KUKA KRL program: MyProgram_150().src

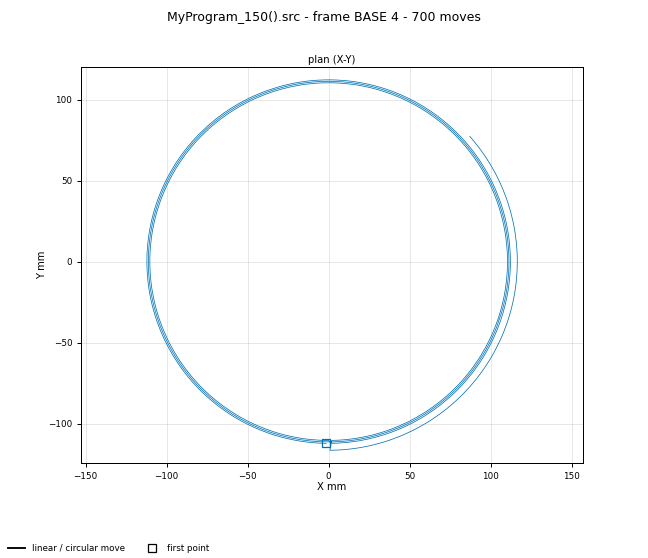
[picture p0: tool path of MyProgram_150().src in frame BASE 4, 700 of 700 moves have a stored position in this frame; points joined in program order, loops and branches not executed]
&ACCESS RVP
&REL 1
&PARAM TEMPLATE = C:\KRC\Roboter\Template\vorgabe
&PARAM EDITMASK = *
DEF MyProgram_150()
; ---- Setting reference (Base) ----
$BASE = BASE_DATA[4]

; --------------------------
; ---- Setting tool (TCP) ----
$TOOL = TOOL_DATA[3]
; --------------------------

$VEL.CP = VEL_APROX_PRINT
Startdeposition()
$VEL.CP = VEL_PRINT
LIN {X -1.5125,Y -112.2052,Z 117,A -94.956,B 24.9546,C -1.5569,E1 24.9968,E2 180.9074} C_DIS
LIN {X -5.7885,Y -112.0653,Z 117,A -97.1016,B 24.9546,C -1.5583,E1 24.9908,E2 183.05} C_DIS
LIN {X -9.0238,Y -111.8506,Z 117,A -99.1979,B 24.9556,C -1.5398,E1 24.9848,E2 185.1911} C_DIS
LIN {X -12.7167,Y -111.4916,Z 117,A -100.657,B 24.9545,C -1.5583,E1 24.9809,E2 186.6072} C_DIS
LIN {X -17.0349,Y -110.9135,Z 117,A -102.8531,B 24.9545,C -1.56,E1 24.9748,E2 188.801} C_DIS
LIN {X -20.6022,Y -110.3083,Z 117,A -104.7565,B 24.9545,C -1.5583,E1 24.9696,E2 190.7105} C_DIS
LIN {X -25.8364,Y -109.2008,Z 117,A -107.366,B 24.9541,C -1.5646,E1 24.9625,E2 193.3082} C_DIS
LIN {X -29.1128,Y -108.3718,Z 117,A -109.2021,B 24.9543,C -1.5611,E1 24.9575,E2 195.1553} C_DIS
LIN {X -32.9964,Y -107.2534,Z 117,A -111.2303,B 24.9542,C -1.564,E1 24.9521,E2 197.18} C_DIS
LIN {X -36.1753,Y -106.2236,Z 117,A -112.94,B 24.9541,C -1.5652,E1 24.9476,E2 198.89} C_DIS
LIN {X -41.7306,Y -104.1678,Z 117,A -116.2554,B 24.9546,C -1.5561,E1 24.9388,E2 202.2341} C_DIS
LIN {X -46.6403,Y -102.0638,Z 117,A -118.7805,B 24.954,C -1.5674,E1 24.9324,E2 204.7384} C_DIS
LIN {X -49.8054,Y -100.5555,Z 117,A -120.8158,B 24.9544,C -1.5596,E1 24.9273,E2 206.7975} C_DIS
LIN {X -53.3163,Y -98.739,Z 117,A -122.531,B 24.9535,C -1.5746,E1 24.9231,E2 208.4819} C_DIS
LIN {X -56.3522,Y -97.0395,Z 117,A -124.7681,B 24.9545,C -1.5584,E1 24.9176,E2 210.7639} C_DIS
LIN {X -59.4233,Y -95.1885,Z 117,A -125.8907,B 24.9526,C -1.5899,E1 24.9151,E2 211.8152} C_DIS
LIN {X -61.8008,Y -93.6624,Z 117,A -127.5917,B 24.9531,C -1.5817,E1 24.911,E2 213.5414} C_DIS
LIN {X -66.4782,Y -90.4029,Z 117,A -130.4958,B 24.9528,C -1.5868,E1 24.9044,E2 216.4431} C_DIS
LIN {X -69.3755,Y -88.1992,Z 117,A -132.4481,B 24.9528,C -1.5864,E1 24.9001,E2 218.4035} C_DIS
LIN {X -72.4947,Y -85.6542,Z 117,A -134.4851,B 24.9526,C -1.5911,E1 24.8957,E2 220.4373} C_DIS
LIN {X -75.0296,Y -83.4422,Z 117,A -136.1776,B 24.9523,C -1.5955,E1 24.8922,E2 222.126} C_DIS
LIN {X -79.2176,Y -79.4784,Z 117,A -139.0952,B 24.9519,C -1.6027,E1 24.8863,E2 225.0385} C_DIS
LIN {X -81.6863,Y -76.9372,Z 117,A -141.3411,B 24.9527,C -1.5894,E1 24.8819,E2 227.3258} C_DIS
LIN {X -84.0515,Y -74.349,Z 117,A -142.6578,B 24.9513,C -1.6121,E1 24.8796,E2 228.5943} C_DIS
LIN {X -86.8434,Y -71.0668,Z 117,A -145.025,B 24.9513,C -1.6107,E1 24.8753,E2 230.9758} C_DIS
LIN {X -89.0383,Y -68.2951,Z 117,A -146.8336,B 24.9511,C -1.6149,E1 24.8722,E2 232.7828} C_DIS
LIN {X -91.2603,Y -65.2959,Z 117,A -148.6799,B 24.9507,C -1.6221,E1 24.8692,E2 234.6212} C_DIS
LIN {X -93.1631,Y -62.5525,Z 117,A -150.6796,B 24.9511,C -1.6148,E1 24.866,E2 236.648} C_DIS
LIN {X -96.2181,Y -57.7447,Z 117,A -153.4338,B 24.9503,C -1.6285,E1 24.862,E2 239.3836} C_DIS
LIN {X -98.0482,Y -54.5762,Z 117,A -155.8431,B 24.9513,C -1.6126,E1 24.8586,E2 241.8434} C_DIS
LIN {X -100.1395,Y -50.6388,Z 117,A -157.3726,B 24.9491,C -1.648,E1 24.8568,E2 243.2969} C_DIS
LIN {X -101.3521,Y -48.166,Z 117,A -158.8369,B 24.9491,C -1.6497,E1 24.855,E2 244.7651} C_DIS
LIN {X -102.7604,Y -45.0816,Z 117,A -160.6671,B 24.9489,C -1.6508,E1 24.8529,E2 246.6026} C_DIS
LIN {X -104.005,Y -42.1305,Z 117,A -162.302,B 24.9486,C -1.6556,E1 24.8511,E2 248.2352} C_DIS
LIN {X -105.7444,Y -37.5537,Z 117,A -164.6186,B 24.9477,C -1.6701,E1 24.8489,E2 250.5302} C_DIS
LIN {X -106.8716,Y -34.2124,Z 117,A -166.8469,B 24.9484,C -1.659,E1 24.8469,E2 252.7979} C_DIS
LIN {X -108.0632,Y -30.2401,Z 117,A -168.866,B 24.9478,C -1.6692,E1 24.8453,E2 254.8042} C_DIS
LIN {X -108.9967,Y -26.6779,Z 117,A -170.6645,B 24.9472,C -1.6782,E1 24.8441,E2 256.5917} C_DIS
LIN {X -109.7546,Y -23.3715,Z 117,A -172.4769,B 24.9471,C -1.6805,E1 24.843,E2 258.4094} C_DIS
LIN {X -110.4905,Y -19.5938,Z 117,A -174.4741,B 24.9468,C -1.6855,E1 24.842,E2 260.4065} C_DIS
LIN {X -111.1169,Y -15.6532,Z 117,A -176.3681,B 24.946,C -1.6975,E1 24.8412,E2 262.2832} C_DIS
LIN {X -111.5012,Y -12.6345,Z 117,A -178.0918,B 24.9461,C -1.6959,E1 24.8407,E2 264.021} C_DIS
LIN {X -111.8621,Y -8.8796,Z 117,A -179.9252,B 24.9455,C -1.7057,E1 24.8402,E2 265.8421} C_DIS
LIN {X -112.1042,Y -4.9643,Z 117,A 178.0019,B 24.9452,C -1.7094,E1 24.8399,E2 267.9185} C_DIS
LIN {X -112.2093,Y -1.0958,Z 117,A 176.0457,B 24.9448,C -1.7166,E1 24.8398,E2 269.8693} C_DIS
LIN {X -112.1374,Y 4.1928,Z 117,A 173.4446,B 24.944,C -1.7292,E1 24.8399,E2 272.4561} C_DIS
LIN {X -112.0034,Y 6.9038,Z 117,A 171.8392,B 24.9442,C -1.7252,E1 24.8402,E2 274.0806} C_DIS
LIN {X -111.7118,Y 10.6091,Z 117,A 169.9421,B 24.9438,C -1.7315,E1 24.8406,E2 275.9742} C_DIS
LIN {X -111.2466,Y 14.7055,Z 117,A 167.8342,B 24.9434,C -1.7382,E1 24.8414,E2 278.0787} C_DIS
LIN {X -110.6476,Y 18.6849,Z 117,A 165.8922,B 24.9427,C -1.7492,E1 24.8422,E2 280.0061} C_DIS
LIN {X -109.9711,Y 22.3248,Z 117,A 163.9291,B 24.9424,C -1.7525,E1 24.8432,E2 281.9729} C_DIS
LIN {X -109.2275,Y 25.721,Z 117,A 162.069,B 24.9423,C -1.7549,E1 24.8444,E2 283.8381} C_DIS
LIN {X -108.2907,Y 29.4132,Z 117,A 160.2595,B 24.9415,C -1.7663,E1 24.8457,E2 285.6309} C_DIS
LIN {X -107.357,Y 32.662,Z 117,A 158.2689,B 24.9418,C -1.7616,E1 24.8473,E2 287.6443} C_DIS
LIN {X -106.3302,Y 35.8592,Z 117,A 156.7529,B 24.941,C -1.7747,E1 24.8486,E2 289.1378} C_DIS
LIN {X -105.2682,Y 38.8689,Z 117,A 155.1631,B 24.9405,C -1.7813,E1 24.8501,E2 290.7209} C_DIS
LIN {X -104.0689,Y 41.9735,Z 117,A 153.3117,B 24.9405,C -1.7807,E1 24.852,E2 292.584} C_DIS
LIN {X -102.6445,Y 45.3475,Z 117,A 150.7978,B 24.9418,C -1.7617,E1 24.8549,E2 295.1569} C_DIS
LIN {X -100.6823,Y 49.5496,Z 117,A 149.0628,B 24.9397,C -1.7931,E1 24.8569,E2 296.8266} C_DIS
LIN {X -98.9283,Y 52.9675,Z 117,A 147.0344,B 24.9395,C -1.7963,E1 24.8595,E2 298.8581} C_DIS
LIN {X -97.1624,Y 56.1383,Z 117,A 145.3017,B 24.9388,C -1.8064,E1 24.8619,E2 300.5758} C_DIS
LIN {X -95.2496,Y 59.3256,Z 117,A 143.0052,B 24.9395,C -1.7965,E1 24.8653,E2 302.9078} C_DIS
LIN {X -93.486,Y 62.0683,Z 117,A 141.5329,B 24.9387,C -1.8086,E1 24.8675,E2 304.3585} C_DIS
LIN {X -91.6074,Y 64.8095,Z 117,A 139.9194,B 24.9382,C -1.8165,E1 24.8701,E2 305.9611} C_DIS
LIN {X -89.6293,Y 67.5174,Z 117,A 137.734,B 24.9391,C -1.8029,E1 24.8739,E2 308.1894} C_DIS
LIN {X -87.2066,Y 70.6186,Z 117,A 136.2751,B 24.9373,C -1.8295,E1 24.8763,E2 309.5917} C_DIS
LIN {X -83.2861,Y 75.204,Z 117,A 133.3752,B 24.9362,C -1.8445,E1 24.8816,E2 312.469} C_DIS
LIN {X -80.5138,Y 78.1644,Z 117,A 130.8616,B 24.9371,C -1.8324,E1 24.8865,E2 315.0226} C_DIS
LIN {X -74.6442,Y 83.7873,Z 117,A 126.8667,B 24.936,C -1.8483,E1 24.8945,E2 318.9959} C_DIS
LIN {X -70.5545,Y 87.2586,Z 117,A 124.4485,B 24.9347,C -1.867,E1 24.8996,E2 321.3788} C_DIS
LIN {X -67.8838,Y 89.354,Z 117,A 122.5036,B 24.935,C -1.8623,E1 24.904,E2 323.342} C_DIS
LIN {X -64.7113,Y 91.6774,Z 117,A 119.9198,B 24.9363,C -1.8438,E1 24.9099,E2 325.9789} C_DIS
LIN {X -61.7752,Y 93.6793,Z 117,A 118.5231,B 24.9349,C -1.8638,E1 24.9131,E2 327.3326} C_DIS
LIN {X -58.5579,Y 95.7239,Z 117,A 116.5933,B 24.9346,C -1.8681,E1 24.9176,E2 329.2582} C_DIS
LIN {X -55.8629,Y 97.3207,Z 117,A 115.0159,B 24.9343,C -1.8719,E1 24.9214,E2 330.8313} C_DIS
LIN {X -52.9912,Y 98.9154,Z 117,A 112.7947,B 24.9356,C -1.8532,E1 24.927,E2 333.1033} C_DIS
LIN {X -49.5821,Y 100.6662,Z 117,A 111.2451,B 24.9343,C -1.8725,E1 24.9308,E2 334.611} C_DIS
LIN {X -45.8433,Y 102.4229,Z 117,A 108.3059,B 24.9363,C -1.8428,E1 24.9385,E2 337.628} C_DIS
LIN {X -40.6091,Y 104.6092,Z 117,A 106.523,B 24.933,C -1.8912,E1 24.9428,E2 339.2998} C_DIS
LIN {X -38.2643,Y 105.4887,Z 117,A 105.0656,B 24.9333,C -1.8857,E1 24.9467,E2 340.7734} C_DIS
LIN {X -30.9788,Y 107.8539,Z 117,A 101.3274,B 24.9325,C -1.8972,E1 24.9566,E2 344.4908} C_DIS
LIN {X -28.4362,Y 108.5525,Z 117,A 99.6995,B 24.9332,C -1.8871,E1 24.961,E2 346.1451} C_DIS
LIN {X -25.1714,Y 109.3544,Z 117,A 97.9354,B 24.9332,C -1.8868,E1 24.9658,E2 347.9122} C_DIS
LIN {X -21.2376,Y 110.186,Z 117,A 96.0146,B 24.9328,C -1.8939,E1 24.971,E2 349.8184} C_DIS
LIN {X -18.1728,Y 110.7332,Z 117,A 94.4475,B 24.9326,C -1.896,E1 24.9753,E2 351.382} C_DIS
LIN {X -13.9046,Y 111.3504,Z 117,A 92.3061,B 24.9323,C -1.8999,E1 24.9812,E2 353.516} C_DIS
LIN {X -9.8507,Y 111.7818,Z 117,A 90.2123,B 24.9323,C -1.9005,E1 24.9871,E2 355.6095} C_DIS
LIN {X -7.0871,Y 111.991,Z 117,A 88.5994,B 24.9328,C -1.8929,E1 24.9916,E2 357.241} C_DIS
LIN {X -2.0943,Y 112.1945,Z 117,A 85.7771,B 24.9336,C -1.8825,E1 24.9996,E2 360.0883} C_DIS
LIN {X 1.2742,Y 112.2083,Z 117,A 84.6091,B 24.9319,C -1.9057,E1 25.0027,E2 361.2014} C_DIS
LIN {X 4.8323,Y 112.1099,Z 117,A 82.6215,B 24.9324,C -1.8988,E1 25.0083,E2 363.2049} C_DIS
LIN {X 9.5577,Y 111.8079,Z 117,A 80.214,B 24.9324,C -1.8991,E1 25.015,E2 365.6106} C_DIS
LIN {X 13.3506,Y 111.4174,Z 117,A 78.1427,B 24.9328,C -1.8936,E1 25.0207,E2 367.6934} C_DIS
LIN {X 17.2419,Y 110.8815,Z 117,A 76.2936,B 24.9324,C -1.8996,E1 25.0258,E2 369.5266} C_DIS
LIN {X 20.1907,Y 110.3831,Z 117,A 74.6472,B 24.9328,C -1.894,E1 25.0304,E2 371.1845} C_DIS
LIN {X 24.2884,Y 109.5546,Z 117,A 72.4808,B 24.9329,C -1.8916,E1 25.0363,E2 373.3538} C_DIS
LIN {X 28.0609,Y 108.6489,Z 117,A 70.6583,B 24.9325,C -1.8972,E1 25.0412,E2 375.1604} C_DIS
LIN {X 31.3668,Y 107.7425,Z 117,A 68.7397,B 24.9331,C -1.8888,E1 25.0464,E2 377.0957} C_DIS
LIN {X 35.0187,Y 106.6111,Z 117,A 66.4582,B 24.9342,C -1.8733,E1 25.0525,E2 379.4097} C_DIS
LIN {X 38.3665,Y 105.4514,Z 117,A 65.4478,B 24.9319,C -1.9057,E1 25.055,E2 380.3413} C_DIS
LIN {X 41.2551,Y 104.3554,Z 117,A 63.4643,B 24.9333,C -1.8867,E1 25.0603,E2 382.3654} C_DIS
LIN {X 44.747,Y 102.9063,Z 117,A 61.6337,B 24.9331,C -1.8889,E1 25.0649,E2 384.1865} C_DIS
LIN {X 49.1094,Y 100.8988,Z 117,A 59.3592,B 24.9328,C -1.8936,E1 25.0707,E2 386.4441} C_DIS
LIN {X 52.9738,Y 98.9248,Z 117,A 55.9431,B 24.9366,C -1.8391,E1 25.0794,E2 389.9793} C_DIS
LIN {X 58.1394,Y 95.9782,Z 117,A 54.0163,B 24.9336,C -1.8823,E1 25.0838,E2 391.798} C_DIS
LIN {X 62.8187,Y 92.9828,Z 117,A 51.1015,B 24.9341,C -1.8744,E1 25.0906,E2 394.7221} C_DIS
LIN {X 65.5667,Y 91.0671,Z 117,A 49.3016,B 24.9346,C -1.8675,E1 25.0947,E2 396.532} C_DIS
LIN {X 68.3874,Y 88.9672,Z 117,A 47.564,B 24.9346,C -1.8668,E1 25.0986,E2 398.2649} C_DIS
LIN {X 71.2508,Y 86.693,Z 117,A 45.6537,B 24.9351,C -1.8614,E1 25.1027,E2 400.1809} C_DIS
LIN {X 74.0379,Y 84.3236,Z 117,A 42.9238,B 24.9379,C -1.8201,E1 25.1087,E2 402.9974} C_DIS
LIN {X 78.3419,Y 80.3427,Z 117,A 40.982,B 24.9352,C -1.8598,E1 25.1124,E2 404.8375} C_DIS
LIN {X 82.243,Y 76.3446,Z 117,A 38.1481,B 24.9355,C -1.8543,E1 25.1179,E2 407.6722} C_DIS
LIN {X 84.3331,Y 74.0269,Z 117,A 36.4291,B 24.9362,C -1.8451,E1 25.1211,E2 409.4052} C_DIS
LIN {X 86.6293,Y 71.3275,Z 117,A 34.2171,B 24.9377,C -1.823,E1 25.1251,E2 411.6592} C_DIS
LIN {X 88.8607,Y 68.5257,Z 117,A 32.8714,B 24.9365,C -1.8399,E1 25.1273,E2 412.9585} C_DIS
LIN {X 91.0579,Y 65.5797,Z 117,A 30.8711,B 24.9372,C -1.8297,E1 25.1306,E2 414.9733} C_DIS
LIN {X 93.2181,Y 62.4712,Z 117,A 28.7974,B 24.938,C -1.8185,E1 25.1339,E2 417.0633} C_DIS
LIN {X 95.3528,Y 59.1603,Z 117,A 26.9952,B 24.9377,C -1.8225,E1 25.1366,E2 418.847} C_DIS
LIN {X 97.6683,Y 55.2565,Z 117,A 24.8595,B 24.9377,C -1.8243,E1 25.1396,E2 420.9673} C_DIS
LIN {X 99.1265,Y 52.5931,Z 117,A 23.2054,B 24.9382,C -1.8154,E1 25.1418,E2 422.6338} C_DIS
LIN {X 100.6594,Y 49.5957,Z 117,A 21.0654,B 24.9398,C -1.7917,E1 25.1445,E2 424.8181} C_DIS
LIN {X 102.2017,Y 46.3343,Z 117,A 19.95,B 24.938,C -1.8191,E1 25.1457,E2 425.8631} C_DIS
LIN {X 103.3763,Y 43.65,Z 117,A 18.0055,B 24.9396,C -1.7945,E1 25.1479,E2 427.8548} C_DIS
LIN {X 105.4616,Y 38.3386,Z 117,A 15.2835,B 24.9396,C -1.7945,E1 25.1506,E2 430.5617} C_DIS
LIN {X 106.7401,Y 34.6199,Z 117,A 13.2706,B 24.9401,C -1.7882,E1 25.1524,E2 432.578} C_DIS
LIN {X 107.7174,Y 31.4513,Z 117,A 11.6079,B 24.9403,C -1.7844,E1 25.1537,E2 434.2402} C_DIS
LIN {X 108.6805,Y 27.9381,Z 117,A 9.7992,B 24.9405,C -1.781,E1 25.155,E2 436.0466} C_DIS
LIN {X 109.5315,Y 24.3944,Z 117,A 7.3036,B 24.9428,C -1.7465,E1 25.1566,E2 438.6089} C_DIS
LIN {X 110.3914,Y 20.1444,Z 117,A 5.9808,B 24.9406,C -1.7799,E1 25.1573,E2 439.8455} C_DIS
LIN {X 111.0865,Y 15.8674,Z 117,A 3.5316,B 24.9418,C -1.762,E1 25.1583,E2 442.3223} C_DIS
LIN {X 111.6731,Y 11.0218,Z 117,A 1.1435,B 24.942,C -1.7588,E1 25.1591,E2 444.704} C_DIS
LIN {X 112.1214,Y 4.5648,Z 117,A -2.0342,B 24.9424,C -1.7539,E1 25.1597,E2 447.8745} C_DIS
LIN {X 112.209,Y -1.1578,Z 117,A -5.5196,B 24.9446,C -1.7187,E1 25.1597,E2 451.4219} C_DIS
LIN {X 112.1246,Y -4.49,Z 117,A -6.586,B 24.9431,C -1.7421,E1 25.1597,E2 452.4269} C_DIS
LIN {X 111.8754,Y -8.7133,Z 117,A -9.5383,B 24.9459,C -1.699,E1 25.1591,E2 455.4631} C_DIS
LIN {X 111.476,Y -12.8504,Z 117,A -11.0335,B 24.9445,C -1.7206,E1 25.1586,E2 456.8988} C_DIS
LIN {X 110.7693,Y -17.9569,Z 117,A -13.5626,B 24.9448,C -1.7167,E1 25.1576,E2 459.4221} C_DIS
LIN {X 110.2165,Y -21.0789,Z 117,A -15.2898,B 24.9454,C -1.7065,E1 25.1567,E2 461.1632} C_DIS
LIN {X 108.8822,Y -27.1473,Z 117,A -18.3294,B 24.9457,C -1.7023,E1 25.1549,E2 464.195} C_DIS
LIN {X 107.6895,Y -31.5453,Z 117,A -21.5658,B 24.9488,C -1.6537,E1 25.1523,E2 467.5275} C_DIS
LIN {X 106.1317,Y -36.4411,Z 117,A -23.6033,B 24.9476,C -1.6719,E1 25.1505,E2 469.5107} C_DIS
LIN {X 104.3708,Y -41.2159,Z 117,A -25.9952,B 24.9476,C -1.6731,E1 25.1482,E2 471.8864} C_DIS
LIN {X 102.7075,Y -45.2029,Z 117,A -27.9869,B 24.9474,C -1.6761,E1 25.146,E2 473.8601} C_DIS
LIN {X 101.6998,Y -47.4252,Z 117,A -29.3518,B 24.9479,C -1.6668,E1 25.1444,E2 475.2394} C_DIS
LIN {X 100.2342,Y -50.4536,Z 117,A -32.1322,B 24.9512,C -1.6138,E1 25.1408,E2 478.13} C_DIS
LIN {X 97.3124,Y -55.8773,Z 117,A -34.1895,B 24.9488,C -1.6535,E1 25.1381,E2 480.0831} C_DIS
LIN {X 95.5736,Y -58.8052,Z 117,A -36.4836,B 24.9506,C -1.6233,E1 25.1347,E2 482.4366} C_DIS
LIN {X 93.3986,Y -62.2009,Z 117,A -37.9027,B 24.9492,C -1.6463,E1 25.1326,E2 483.7944} C_DIS
LIN {X 90.3118,Y -66.6026,Z 117,A -40.7755,B 24.95,C -1.6329,E1 25.1279,E2 486.6849} C_DIS
LIN {X 87.8329,Y -69.8386,Z 117,A -42.8903,B 24.9505,C -1.6258,E1 25.1243,E2 488.8066} C_DIS
LIN {X 85.434,Y -72.7531,Z 117,A -44.7029,B 24.9505,C -1.6258,E1 25.121,E2 490.6106} C_DIS
LIN {X 82.4378,Y -76.1323,Z 117,A -46.96,B 24.9507,C -1.6221,E1 25.1168,E2 492.8665} C_DIS
LIN {X 79.3195,Y -79.3776,Z 117,A -49.1838,B 24.9508,C -1.6197,E1 25.1125,E2 495.0865} C_DIS
LIN {X 76.5096,Y -82.0885,Z 117,A -51.5205,B 24.9521,C -1.5995,E1 25.1077,E2 497.4611} C_DIS
LIN {X 72.9345,Y -85.2794,Z 117,A -53.8887,B 24.9521,C -1.5974,E1 25.1027,E2 499.825} C_DIS
LIN {X 69.0668,Y -88.4431,Z 117,A -56.5691,B 24.9529,C -1.586,E1 25.0968,E2 502.5224} C_DIS
LIN {X 64.2774,Y -91.9808,Z 117,A -58.9994,B 24.9516,C -1.6068,E1 25.0915,E2 504.8949} C_DIS
LIN {X 59.4079,Y -95.1982,Z 117,A -62.5891,B 24.9536,C -1.5739,E1 25.0829,E2 508.5506} C_DIS
LIN {X 56.5135,Y -96.9468,Z 117,A -63.8758,B 24.9526,C -1.5901,E1 25.0799,E2 509.7952} C_DIS
LIN {X 53.8026,Y -98.4752,Z 117,A -66.4463,B 24.9553,C -1.5443,E1 25.0734,E2 512.4665} C_DIS
LIN {X 48.7959,Y -101.0494,Z 117,A -68.3984,B 24.9532,C -1.5798,E1 25.0687,E2 514.3293} C_DIS
LIN {X 45.5629,Y -102.5493,Z 117,A -70.3942,B 24.9539,C -1.5692,E1 25.0636,E2 516.3451} C_DIS
LIN {X 41.3238,Y -104.3285,Z 117,A -72.3071,B 24.9529,C -1.5849,E1 25.0588,E2 518.2165} C_DIS
LIN {X 38.0018,Y -105.5844,Z 117,A -74.2648,B 24.9535,C -1.5761,E1 25.0536,E2 520.1909} C_DIS
LIN {X 35.0271,Y -106.6084,Z 117,A -76.0262,B 24.954,C -1.5673,E1 25.0489,E2 521.9698} C_DIS
LIN {X 31.2217,Y -107.7851,Z 117,A -77.9011,B 24.9537,C -1.5719,E1 25.0439,E2 523.8306} C_DIS
LIN {X 28.1952,Y -108.6144,Z 117,A -79.6196,B 24.9541,C -1.5651,E1 25.0392,E2 525.5623} C_DIS
LIN {X 24.5867,Y -109.4895,Z 117,A -82.3539,B 24.9563,C -1.5273,E1 25.0316,E2 528.3825} C_DIS
LIN {X 19.2447,Y -110.5532,Z 117,A -84.1695,B 24.954,C -1.5664,E1 25.0268,E2 530.1034} C_DIS
LIN {X 16.6494,Y -110.9731,Z 117,A -85.6308,B 24.9544,C -1.5603,E1 25.0228,E2 531.5779} C_DIS
LIN {X 10.8762,Y -111.6871,Z 117,A -88.4781,B 24.9542,C -1.5637,E1 25.0149,E2 534.4149} C_DIS
LIN {X 5.3933,Y -112.0858,Z 117,A -91.2425,B 24.9542,C -1.5643,E1 25.0072,E2 537.1768} C_DIS
LIN {X 2.3796,Y -112.1892,Z 117,A -93.4048,B 24.9557,C -1.5374,E1 25.001,E2 539.4024} C_DIS
LIN {X 2.3796,Y -112.1892,Z 117,A -93.4048,B 24.9557,C -1.5374,E1 25.001,E2 539.4024} C_DIS
Enddeposition()
LIN {X 0.7912,Y -111.3047,Z 117,A -93.2213,B 24.9523,C -1.5953,E1 25.0019,E2 539.0817} C_DIS
Startdeposition()
$VEL.CP = VEL_PRINT
LIN {X 3.6719,Y -111.2517,Z 117,A -91.467,B 24.9516,C -1.6073,E1 25.0068,E2 537.2993} C_DIS
LIN {X 7.3807,Y -111.0671,Z 117,A -89.4219,B 24.9512,C -1.6139,E1 25.0126,E2 535.2394} C_DIS
LIN {X 11.965,Y -110.6677,Z 117,A -87.0248,B 24.951,C -1.6164,E1 25.0193,E2 532.8379} C_DIS
LIN {X 16.0589,Y -110.1482,Z 117,A -85.021,B 24.9513,C -1.6126,E1 25.0248,E2 530.8448} C_DIS
LIN {X 19.6319,Y -109.5671,Z 117,A -83.1834,B 24.9513,C -1.6129,E1 25.0298,E2 529.0082} C_DIS
LIN {X 24.4922,Y -108.5855,Z 117,A -80.6381,B 24.9511,C -1.6149,E1 25.0368,E2 526.4615} C_DIS
LIN {X 27.696,Y -107.8113,Z 117,A -78.9839,B 24.9511,C -1.6148,E1 25.0413,E2 524.8101} C_DIS
LIN {X 31.3626,Y -106.8028,Z 117,A -77.2198,B 24.9515,C -1.6085,E1 25.046,E2 523.0638} C_DIS
LIN {X 35.1289,Y -105.6244,Z 117,A -75.0006,B 24.9509,C -1.6192,E1 25.0519,E2 520.8235} C_DIS
LIN {X 40.2173,Y -103.794,Z 117,A -72.2803,B 24.9509,C -1.6201,E1 25.059,E2 518.1067} C_DIS
LIN {X 45.1793,Y -101.7327,Z 117,A -69.3746,B 24.9502,C -1.6303,E1 25.0666,E2 515.1836} C_DIS
LIN {X 48.5531,Y -100.1654,Z 117,A -67.7006,B 24.9507,C -1.6228,E1 25.0707,E2 513.5318} C_DIS
LIN {X 51.8036,Y -98.5228,Z 117,A -65.7093,B 24.9501,C -1.6311,E1 25.0757,E2 511.5263} C_DIS
LIN {X 54.7137,Y -96.9382,Z 117,A -64.0643,B 24.9501,C -1.6314,E1 25.0797,E2 509.8853} C_DIS
LIN {X 57.4854,Y -95.3201,Z 117,A -62.4047,B 24.9499,C -1.6348,E1 25.0837,E2 508.2228} C_DIS
LIN {X 59.6849,Y -93.9593,Z 117,A -60.5223,B 24.9482,C -1.6621,E1 25.0883,E2 506.2821} C_DIS
LIN {X 62.9107,Y -91.8312,Z 117,A -58.8648,B 24.9489,C -1.6512,E1 25.092,E2 504.656} C_DIS
LIN {X 68.1884,Y -87.9818,Z 117,A -55.6621,B 24.9489,C -1.6512,E1 25.0992,E2 501.4647} C_DIS
LIN {X 70.9844,Y -85.7415,Z 117,A -53.7155,B 24.9484,C -1.6599,E1 25.1034,E2 499.505} C_DIS
LIN {X 73.8261,Y -83.3089,Z 117,A -51.9046,B 24.9484,C -1.6592,E1 25.1072,E2 497.7029} C_DIS
LIN {X 76.14,Y -81.1978,Z 117,A -50.3167,B 24.9482,C -1.6619,E1 25.1105,E2 496.115} C_DIS
LIN {X 78.9755,Y -78.4431,Z 117,A -48.4588,B 24.9484,C -1.6589,E1 25.1141,E2 494.272} C_DIS
LIN {X 81.2337,Y -76.1018,Z 117,A -46.8398,B 24.9484,C -1.6606,E1 25.1172,E2 492.656} C_DIS
LIN {X 83.1471,Y -74.0069,Z 117,A -45.1503,B 24.9474,C -1.6747,E1 25.1204,E2 490.9407} C_DIS
LIN {X 85.4358,Y -71.3523,Z 117,A -43.5596,B 24.9478,C -1.6698,E1 25.1233,E2 489.3689} C_DIS
LIN {X 88.1374,Y -67.9864,Z 117,A -41.2591,B 24.9472,C -1.6793,E1 25.1273,E2 487.0567} C_DIS
LIN {X 90.2267,Y -65.1888,Z 117,A -38.7461,B 24.9448,C -1.717,E1 25.1316,E2 484.4669} C_DIS
LIN {X 92.8033,Y -61.4651,Z 117,A -36.82,B 24.9455,C -1.705,E1 25.1345,E2 482.5786} C_DIS
LIN {X 95.3166,Y -57.4913,Z 117,A -34.6168,B 24.9457,C -1.7021,E1 25.1377,E2 480.3936} C_DIS
LIN {X 97.1438,Y -54.3455,Z 117,A -32.8682,B 24.9457,C -1.7019,E1 25.1401,E2 478.6544} C_DIS
LIN {X 99.4284,Y -50.0481,Z 117,A -30.3408,B 24.9452,C -1.7104,E1 25.1434,E2 476.1204} C_DIS
LIN {X 100.7054,Y -47.4238,Z 117,A -28.7823,B 24.9447,C -1.7175,E1 25.1452,E2 474.5534} C_DIS
LIN {X 102.2779,Y -43.9313,Z 117,A -26.3702,B 24.943,C -1.7438,E1 25.148,E2 472.0925} C_DIS
LIN {X 103.7299,Y -40.3805,Z 117,A -24.8415,B 24.9439,C -1.7295,E1 25.1495,E2 470.6061} C_DIS
LIN {X 106.8436,Y -31.2251,Z 117,A -19.9672,B 24.9432,C -1.7403,E1 25.1538,E2 465.7339} C_DIS
LIN {X 107.6845,Y -28.1895,Z 117,A -18.2548,B 24.9426,C -1.7497,E1 25.155,E2 464.0092} C_DIS
LIN {X 108.7371,Y -23.8035,Z 117,A -16.0947,B 24.9426,C -1.7497,E1 25.1563,E2 461.8614} C_DIS
LIN {X 109.4401,Y -20.3379,Z 117,A -14.1325,B 24.9418,C -1.7621,E1 25.1574,E2 459.8816} C_DIS
LIN {X 110.0941,Y -16.4313,Z 117,A -12.1143,B 24.9414,C -1.7678,E1 25.1583,E2 457.8618} C_DIS
LIN {X 110.5764,Y -12.7764,Z 117,A -10.5265,B 24.942,C -1.7598,E1 25.1588,E2 456.3023} C_DIS
LIN {X 110.8989,Y -9.6012,Z 117,A -8.632,B 24.9408,C -1.7766,E1 25.1593,E2 454.3793} C_DIS
LIN {X 111.1556,Y -5.9024,Z 117,A -6.8359,B 24.9408,C -1.7777,E1 25.1596,E2 452.5913} C_DIS
LIN {X 111.2856,Y -2.4566,Z 117,A -5.2566,B 24.941,C -1.7746,E1 25.1598,E2 451.0288} C_DIS
LIN {X 111.3125,Y 0.0831,Z 117,A -3.5658,B 24.9395,C -1.7964,E1 25.1598,E2 449.2967} C_DIS
LIN {X 111.2115,Y 4.7279,Z 117,A -1.3955,B 24.9397,C -1.794,E1 25.1596,E2 447.1448} C_DIS
LIN {X 110.873,Y 9.8821,Z 117,A 1.2832,B 24.939,C -1.8035,E1 25.159,E2 444.4597} C_DIS
LIN {X 110.5282,Y 13.1884,Z 117,A 3.0465,B 24.9385,C -1.8114,E1 25.1585,E2 442.6883} C_DIS
LIN {X 110.1103,Y 16.3258,Z 117,A 4.6318,B 24.9383,C -1.8145,E1 25.1579,E2 441.1048} C_DIS
LIN {X 109.4586,Y 20.235,Z 117,A 6.5236,B 24.9383,C -1.8142,E1 25.1569,E2 439.2248} C_DIS
LIN {X 108.699,Y 23.9782,Z 117,A 8.6375,B 24.9374,C -1.8272,E1 25.1557,E2 437.0928} C_DIS
LIN {X 107.9345,Y 27.2169,Z 117,A 10.1911,B 24.9376,C -1.8252,E1 25.1547,E2 435.5528} C_DIS
LIN {X 107.1087,Y 30.2998,Z 117,A 11.8751,B 24.9371,C -1.8322,E1 25.1534,E2 433.862} C_DIS
LIN {X 106.0311,Y 33.8811,Z 117,A 13.771,B 24.9368,C -1.8367,E1 25.1519,E2 431.9662} C_DIS
LIN {X 105.1764,Y 36.4481,Z 117,A 15.2594,B 24.9362,C -1.8452,E1 25.1505,E2 430.4661} C_DIS
LIN {X 104.1726,Y 39.2232,Z 117,A 17.2142,B 24.9345,C -1.8696,E1 25.1486,E2 428.4646} C_DIS
LIN {X 102.7181,Y 42.8892,Z 117,A 18.7399,B 24.9357,C -1.8526,E1 25.147,E2 426.9875} C_DIS
LIN {X 101.2541,Y 46.2416,Z 117,A 20.5101,B 24.9357,C -1.8529,E1 25.145,E2 425.2262} C_DIS
LIN {X 99.8083,Y 49.2817,Z 117,A 22.2548,B 24.9353,C -1.8584,E1 25.1429,E2 423.478} C_DIS
LIN {X 98.4926,Y 51.861,Z 117,A 23.645,B 24.9353,C -1.858,E1 25.1411,E2 422.096} C_DIS
LIN {X 97.4235,Y 53.8448,Z 117,A 25.0003,B 24.9345,C -1.87,E1 25.1392,E2 420.7195} C_DIS
LIN {X 94.7192,Y 58.4721,Z 117,A 27.7589,B 24.9339,C -1.8774,E1 25.1353,E2 417.9577} C_DIS
LIN {X 92.6887,Y 61.6389,Z 117,A 29.5429,B 24.9341,C -1.8756,E1 25.1326,E2 416.1867} C_DIS
LIN {X 91.1229,Y 63.9312,Z 117,A 31.105,B 24.9334,C -1.8852,E1 25.1301,E2 414.6096} C_DIS
LIN {X 89.1594,Y 66.641,Z 117,A 32.7447,B 24.9334,C -1.8858,E1 25.1274,E2 412.9764} C_DIS
LIN {X 86.87,Y 69.6014,Z 117,A 34.7547,B 24.9327,C -1.8942,E1 25.1239,E2 410.956} C_DIS
LIN {X 84.8355,Y 72.0647,Z 117,A 36.2507,B 24.9329,C -1.8915,E1 25.1212,E2 409.4733} C_DIS
LIN {X 82.7357,Y 74.4664,Z 117,A 37.9869,B 24.9324,C -1.8994,E1 25.118,E2 407.7261} C_DIS
LIN {X 80.603,Y 76.772,Z 117,A 39.7726,B 24.9316,C -1.9105,E1 25.1145,E2 405.922} C_DIS
LIN {X 77.072,Y 80.3139,Z 117,A 42.031,B 24.9322,C -1.902,E1 25.1101,E2 403.6932} C_DIS
LIN {X 73.6095,Y 83.5001,Z 117,A 44.5577,B 24.9315,C -1.9115,E1 25.1048,E2 401.154} C_DIS
LIN {X 70.8644,Y 85.8413,Z 117,A 46.4439,B 24.9311,C -1.9164,E1 25.1008,E2 399.2636} C_DIS
LIN {X 68.2646,Y 87.9231,Z 117,A 48.155,B 24.9309,C -1.9194,E1 25.097,E2 397.5517} C_DIS
LIN {X 64.996,Y 90.3662,Z 117,A 50.0937,B 24.9312,C -1.916,E1 25.0927,E2 395.628} C_DIS
LIN {X 62.9281,Y 91.8194,Z 117,A 51.3594,B 24.9312,C -1.9167,E1 25.0898,E2 394.3651} C_DIS
LIN {X 60.1952,Y 93.6317,Z 117,A 53.1906,B 24.9305,C -1.9257,E1 25.0855,E2 392.5187} C_DIS
LIN {X 56.6394,Y 95.8245,Z 117,A 55.2504,B 24.9305,C -1.925,E1 25.0806,E2 390.4669} C_DIS
LIN {X 51.8967,Y 98.4738,Z 117,A 58.0837,B 24.9301,C -1.9304,E1 25.0736,E2 387.6289} C_DIS
LIN {X 48.4401,Y 100.2196,Z 117,A 60.1484,B 24.9297,C -1.936,E1 25.0684,E2 385.5565} C_DIS
LIN {X 44.6008,Y 101.986,Z 117,A 62.2231,B 24.9299,C -1.9342,E1 25.0632,E2 383.4912} C_DIS
LIN {X 41.8564,Y 103.1427,Z 117,A 63.6756,B 24.9299,C -1.9323,E1 25.0594,E2 382.0465} C_DIS
LIN {X 38.0397,Y 104.6104,Z 117,A 65.8462,B 24.9296,C -1.9372,E1 25.0537,E2 379.8691} C_DIS
LIN {X 33.6778,Y 106.0969,Z 117,A 68.3262,B 24.9292,C -1.9438,E1 25.0471,E2 377.3783} C_DIS
LIN {X 29.708,Y 107.2764,Z 117,A 70.4382,B 24.9292,C -1.9444,E1 25.0415,E2 375.2683} C_DIS
LIN {X 26.3871,Y 108.1391,Z 117,A 72.1271,B 24.9292,C -1.9422,E1 25.0369,E2 373.5871} C_DIS
LIN {X 22.6097,Y 108.9918,Z 117,A 74.1122,B 24.9292,C -1.9429,E1 25.0315,E2 371.6031} C_DIS
LIN {X 19.0352,Y 109.6744,Z 117,A 76.0184,B 24.9291,C -1.945,E1 25.0263,E2 369.694} C_DIS
LIN {X 15.4307,Y 110.2375,Z 117,A 77.9338,B 24.9289,C -1.9471,E1 25.021,E2 367.7753} C_DIS
LIN {X 12.1015,Y 110.6534,Z 117,A 79.4848,B 24.9294,C -1.94,E1 25.0167,E2 366.2423} C_DIS
LIN {X 8.6904,Y 110.9723,Z 117,A 81.3145,B 24.9292,C -1.9429,E1 25.0116,E2 364.4066} C_DIS
LIN {X 5.2151,Y 111.1906,Z 117,A 83.2703,B 24.9287,C -1.9497,E1 25.0061,E2 362.4354} C_DIS
LIN {X 1.5061,Y 111.3031,Z 117,A 85.1829,B 24.9287,C -1.9496,E1 25.0008,E2 360.5234} C_DIS
LIN {X -1.2857,Y 111.3062,Z 117,A 86.5468,B 24.929,C -1.9462,E1 24.997,E2 359.1676} C_DIS
LIN {X -5.244,Y 111.1893,Z 117,A 88.4519,B 24.9294,C -1.94,E1 24.9917,E2 357.2767} C_DIS
LIN {X -8.6503,Y 110.9756,Z 117,A 90.1868,B 24.9296,C -1.9384,E1 24.9869,E2 355.5451} C_DIS
LIN {X -11.4933,Y 110.7171,Z 117,A 91.7672,B 24.9293,C -1.9422,E1 24.9825,E2 353.9547} C_DIS
LIN {X -14.5312,Y 110.3596,Z 117,A 93.4458,B 24.929,C -1.9456,E1 24.9778,E2 352.267} C_DIS
LIN {X -18.0105,Y 109.8458,Z 117,A 94.9541,B 24.93,C -1.9319,E1 24.9737,E2 350.7898} C_DIS
LIN {X -21.2277,Y 109.2693,Z 117,A 96.8396,B 24.9295,C -1.9389,E1 24.9685,E2 348.8857} C_DIS
LIN {X -24.3599,Y 108.6157,Z 117,A 98.5825,B 24.9293,C -1.9414,E1 24.9637,E2 347.1348} C_DIS
LIN {X -27.8869,Y 107.7623,Z 117,A 100.3504,B 24.9298,C -1.9355,E1 24.9589,E2 345.3784} C_DIS
LIN {X -31.3608,Y 106.8033,Z 117,A 102.6009,B 24.9287,C -1.9496,E1 24.9528,E2 343.0907} C_DIS
LIN {X -34.5247,Y 105.8228,Z 117,A 103.8711,B 24.9302,C -1.9299,E1 24.9496,E2 341.865} C_DIS
LIN {X -37.822,Y 104.6899,Z 117,A 105.7612,B 24.9301,C -1.9315,E1 24.9446,E2 339.9674} C_DIS
LIN {X -41.0864,Y 103.4526,Z 117,A 107.6231,B 24.9301,C -1.9317,E1 24.9397,E2 338.1012} C_DIS
LIN {X -46.0334,Y 101.3479,Z 117,A 110.391,B 24.9303,C -1.9276,E1 24.9326,E2 335.3363} C_DIS
LIN {X -48.9912,Y 99.9523,Z 117,A 112.175,B 24.9303,C -1.9289,E1 24.9281,E2 333.5445} C_DIS
LIN {X -52.4246,Y 98.1958,Z 117,A 114.1428,B 24.9305,C -1.9249,E1 24.9233,E2 331.5809} C_DIS
LIN {X -56.0083,Y 96.1968,Z 117,A 116.2111,B 24.9309,C -1.9194,E1 24.9183,E2 329.5197} C_DIS
LIN {X -59.0199,Y 94.3769,Z 117,A 117.9331,B 24.9314,C -1.9124,E1 24.9142,E2 327.8087} C_DIS
LIN {X -61.6857,Y 92.6578,Z 117,A 119.5984,B 24.9316,C -1.9105,E1 24.9103,E2 326.1425} C_DIS
LIN {X -64.4499,Y 90.7558,Z 117,A 121.2943,B 24.9319,C -1.9058,E1 24.9064,E2 324.452} C_DIS
LIN {X -67.3014,Y 88.6633,Z 117,A 123.1703,B 24.932,C -1.9042,E1 24.9022,E2 322.5733} C_DIS
LIN {X -69.9146,Y 86.6161,Z 117,A 124.8883,B 24.9323,C -1.9009,E1 24.8985,E2 320.8568} C_DIS
LIN {X -73.6175,Y 83.4931,Z 117,A 127.4527,B 24.9325,C -1.898,E1 24.8931,E2 318.2893} C_DIS
LIN {X -76.2754,Y 81.0705,Z 117,A 129.2347,B 24.933,C -1.8909,E1 24.8894,E2 316.5168} C_DIS
LIN {X -79.5545,Y 77.8569,Z 117,A 131.9726,B 24.9323,C -1.8999,E1 24.884,E2 313.7458} C_DIS
LIN {X -81.8059,Y 75.4867,Z 117,A 133.3258,B 24.9336,C -1.8827,E1 24.8815,E2 312.4277} C_DIS
LIN {X -84.2391,Y 72.7633,Z 117,A 135.1089,B 24.9342,C -1.8741,E1 24.8782,E2 310.6571} C_DIS
LIN {X -87.3268,Y 69.0245,Z 117,A 137.8263,B 24.934,C -1.8762,E1 24.8734,E2 307.9221} C_DIS
LIN {X -89.507,Y 66.1748,Z 117,A 139.5892,B 24.9346,C -1.8678,E1 24.8705,E2 306.1706} C_DIS
LIN {X -91.5331,Y 63.3412,Z 117,A 141.4296,B 24.9348,C -1.8647,E1 24.8675,E2 304.3285} C_DIS
LIN {X -93.3811,Y 60.5855,Z 117,A 143.1787,B 24.935,C -1.8615,E1 24.8648,E2 302.5783} C_DIS
LIN {X -95.504,Y 57.1816,Z 117,A 145.2467,B 24.9354,C -1.8557,E1 24.8618,E2 300.5136} C_DIS
LIN {X -97.2516,Y 54.1526,Z 117,A 146.9419,B 24.9361,C -1.8464,E1 24.8595,E2 298.8317} C_DIS
LIN {X -98.9848,Y 50.916,Z 117,A 148.7983,B 24.9366,C -1.8395,E1 24.8571,E2 296.9819} C_DIS
LIN {X -100.8417,Y 47.131,Z 117,A 151.026,B 24.9369,C -1.8352,E1 24.8544,E2 294.7524} C_DIS
LIN {X -102.258,Y 43.9767,Z 117,A 152.898,B 24.937,C -1.8333,E1 24.8523,E2 292.8746} C_DIS
LIN {X -103.7867,Y 40.2357,Z 117,A 154.8415,B 24.9378,C -1.8216,E1 24.8503,E2 290.9481} C_DIS
LIN {X -104.9705,Y 37.035,Z 117,A 156.7246,B 24.9378,C -1.821,E1 24.8485,E2 289.0558} C_DIS
LIN {X -106.0405,Y 33.8519,Z 117,A 158.351,B 24.9385,C -1.8116,E1 24.8471,E2 287.4425} C_DIS
LIN {X -107.0074,Y 30.6575,Z 117,A 160.1845,B 24.9385,C -1.8106,E1 24.8456,E2 285.6007} C_DIS
LIN {X -107.9563,Y 27.1319,Z 117,A 162.1585,B 24.9387,C -1.8083,E1 24.8443,E2 283.6208} C_DIS
LIN {X -108.8912,Y 23.0966,Z 117,A 164.297,B 24.9392,C -1.8017,E1 24.843,E2 281.4855} C_DIS
LIN {X -109.4629,Y 20.2114,Z 117,A 165.7938,B 24.9395,C -1.7961,E1 24.8422,E2 279.9931} C_DIS
LIN {X -110.0317,Y 16.8349,Z 117,A 167.4806,B 24.9401,C -1.7875,E1 24.8415,E2 278.3168} C_DIS
LIN {X -110.5109,Y 13.3359,Z 117,A 169.139,B 24.9409,C -1.7754,E1 24.8409,E2 276.6773} C_DIS
LIN {X -110.8451,Y 10.1837,Z 117,A 171.0122,B 24.9407,C -1.7795,E1 24.8403,E2 274.7832} C_DIS
LIN {X -111.1344,Y 6.2858,Z 117,A 172.7936,B 24.9417,C -1.764,E1 24.84,E2 273.0279} C_DIS
LIN {X -111.2583,Y 3.4555,Z 117,A 174.5937,B 24.9411,C -1.7725,E1 24.8398,E2 271.1968} C_DIS
LIN {X -111.3097,Y -0.6131,Z 117,A 176.5814,B 24.9418,C -1.7616,E1 24.8398,E2 269.2231} C_DIS
LIN {X -111.2465,Y -3.8417,Z 117,A 178.2384,B 24.9422,C -1.756,E1 24.8399,E2 267.5696} C_DIS
LIN {X -111.0644,Y -7.4196,Z 117,A -179.9212,B 24.9426,C -1.7499,E1 24.8402,E2 265.7325} C_DIS
LIN {X -110.7742,Y -10.9473,Z 117,A -177.9359,B 24.9426,C -1.7503,E1 24.8407,E2 263.7342} C_DIS
LIN {X -110.4237,Y -14.037,Z 117,A -176.5128,B 24.9434,C -1.7384,E1 24.8412,E2 262.3312} C_DIS
LIN {X -110.0054,Y -17.0046,Z 117,A -174.8611,B 24.9434,C -1.7377,E1 24.8419,E2 260.6713} C_DIS
LIN {X -109.341,Y -20.8551,Z 117,A -172.8762,B 24.9439,C -1.7303,E1 24.8429,E2 258.6922} C_DIS
LIN {X -108.6094,Y -24.389,Z 117,A -170.99,B 24.9442,C -1.7256,E1 24.844,E2 256.8062} C_DIS
LIN {X -107.8183,Y -27.6689,Z 117,A -169.0834,B 24.9442,C -1.7269,E1 24.8453,E2 254.8854} C_DIS
LIN {X -106.687,Y -31.7528,Z 117,A -166.2563,B 24.9429,C -1.7456,E1 24.8476,E2 251.9972} C_DIS
LIN {X -105.1288,Y -36.5837,Z 117,A -164.4526,B 24.9455,C -1.7059,E1 24.8491,E2 250.278} C_DIS
LIN {X -103.8379,Y -40.1055,Z 117,A -162.5395,B 24.9459,C -1.6995,E1 24.851,E2 248.3694} C_DIS
LIN {X -102.7983,Y -42.6988,Z 117,A -160.9169,B 24.9457,C -1.7025,E1 24.8527,E2 246.7306} C_DIS
LIN {X -101.2317,Y -46.2911,Z 117,A -158.8998,B 24.9461,C -1.6967,E1 24.855,E2 244.7162} C_DIS
LIN {X -99.7356,Y -49.4283,Z 117,A -157.4178,B 24.9471,C -1.6796,E1 24.8568,E2 243.2669} C_DIS
LIN {X -98.2537,Y -52.3146,Z 117,A -155.4619,B 24.9467,C -1.6862,E1 24.8594,E2 241.2849} C_DIS
LIN {X -96.5231,Y -55.4405,Z 117,A -153.6455,B 24.9471,C -1.6803,E1 24.8618,E2 239.473} C_DIS
LIN {X -94.5171,Y -58.7955,Z 117,A -151.6407,B 24.9474,C -1.6747,E1 24.8647,E2 237.4713} C_DIS
LIN {X -92.871,Y -61.3624,Z 117,A -149.9662,B 24.9474,C -1.6747,E1 24.8673,E2 235.7882} C_DIS
LIN {X -90.6363,Y -64.6174,Z 117,A -148.0609,B 24.9481,C -1.6646,E1 24.8703,E2 233.8979} C_DIS
LIN {X -88.7214,Y -67.2241,Z 117,A -146.2438,B 24.948,C -1.6665,E1 24.8734,E2 232.0674} C_DIS
LIN {X -86.3641,Y -70.2255,Z 117,A -144.3866,B 24.9485,C -1.6575,E1 24.8766,E2 230.2228} C_DIS
LIN {X -83.7964,Y -73.2702,Z 117,A -142.3877,B 24.9489,C -1.6507,E1 24.8802,E2 228.2311} C_DIS
LIN {X -81.465,Y -75.8559,Z 117,A -140.4275,B 24.9488,C -1.6534,E1 24.884,E2 226.2558} C_DIS
LIN {X -78.7528,Y -78.6686,Z 117,A -138.539,B 24.9493,C -1.6441,E1 24.8876,E2 224.3813} C_DIS
LIN {X -75.8558,Y -81.4651,Z 117,A -136.3944,B 24.9494,C -1.6427,E1 24.892,E2 222.2313} C_DIS
LIN {X -73.4138,Y -83.671,Z 117,A -134.7036,B 24.9496,C -1.6393,E1 24.8955,E2 220.5419} C_DIS
LIN {X -70.7215,Y -85.96,Z 117,A -132.7793,B 24.9496,C -1.64,E1 24.8997,E2 218.6085} C_DIS
LIN {X -67.9357,Y -88.1765,Z 117,A -131.0768,B 24.9501,C -1.6314,E1 24.9034,E2 216.9201} C_DIS
LIN {X -64.3762,Y -90.8085,Z 117,A -128.8114,B 24.9504,C -1.6269,E1 24.9085,E2 214.6575} C_DIS
LIN {X -61.3983,Y -92.8473,Z 117,A -126.9043,B 24.9504,C -1.6259,E1 24.9129,E2 212.7464} C_DIS
LIN {X -58.3219,Y -94.8118,Z 117,A -125.0142,B 24.9506,C -1.6235,E1 24.9174,E2 210.8562} C_DIS
LIN {X -54.9655,Y -96.796,Z 117,A -122.9064,B 24.9506,C -1.6248,E1 24.9225,E2 208.739} C_DIS
LIN {X -51.872,Y -98.4868,Z 117,A -121.1792,B 24.9509,C -1.6188,E1 24.9267,E2 207.0212} C_DIS
LIN {X -48.3754,Y -100.2507,Z 117,A -119.2347,B 24.9512,C -1.6133,E1 24.9316,E2 205.0845} C_DIS
LIN {X -46.1677,Y -101.2873,Z 117,A -118.0658,B 24.9515,C -1.6083,E1 24.9345,E2 203.9246} C_DIS
LIN {X -43.1747,Y -102.5978,Z 117,A -116.196,B 24.9512,C -1.6143,E1 24.9393,E2 202.0363} C_DIS
LIN {X -39.5289,Y -104.0569,Z 117,A -113.9738,B 24.9508,C -1.6207,E1 24.9452,E2 199.7941} C_DIS
LIN {X -35.5802,Y -105.4723,Z 117,A -112.0487,B 24.9515,C -1.6091,E1 24.9502,E2 197.8928} C_DIS
LIN {X -32.0924,Y -106.5863,Z 117,A -110.2336,B 24.9517,C -1.6048,E1 24.955,E2 196.0849} C_DIS
LIN {X -29.042,Y -107.4566,Z 117,A -108.502,B 24.9516,C -1.6078,E1 24.9597,E2 194.3432} C_DIS
LIN {X -25.3484,Y -108.3877,Z 117,A -106.7875,B 24.9522,C -1.5964,E1 24.9643,E2 192.6534} C_DIS
LIN {X -22.5806,Y -108.9978,Z 117,A -105.1495,B 24.9518,C -1.6033,E1 24.9688,E2 190.9972} C_DIS
LIN {X -18.4759,Y -109.768,Z 117,A -102.9995,B 24.9518,C -1.6025,E1 24.9747,E2 188.8467} C_DIS
LIN {X -15.8059,Y -110.1842,Z 117,A -101.4558,B 24.9515,C -1.6087,E1 24.979,E2 187.2872} C_DIS
LIN {X -11.6245,Y -110.7033,Z 117,A -99.324,B 24.9516,C -1.6068,E1 24.9849,E2 185.1584} C_DIS
LIN {X -8.0569,Y -111.0214,Z 117,A -97.4638,B 24.9516,C -1.6074,E1 24.9901,E2 183.296} C_DIS
LIN {X -4.6098,Y -111.2166,Z 117,A -95.7079,B 24.9516,C -1.6067,E1 24.995,E2 181.5414} C_DIS
LIN {X -1.0085,Y -111.3079,Z 117,A -94.1227,B 24.9523,C -1.5955,E1 24.9994,E2 179.9825} C_DIS
LIN {X 0.7912,Y -111.3047,Z 117,A -93.2201,B 24.9523,C -1.5948,E1 25.0019,E2 179.0817} C_DIS
Enddeposition()
LIN {X 0.7912,Y -111.3047,Z 117,A -93.2201,B 24.9523,C -1.5948,E1 25.0019,E2 179.0817} C_DIS
Startdeposition()
$VEL.CP = VEL_PRINT
LIN {X -0.0318,Y -110.4118,Z 117,A -94.1173,B 24.9526,C -1.5905,E1 24.9993,E2 179.9889} C_DIS
LIN {X -2.422,Y -110.384,Z 117,A -95.4038,B 24.9527,C -1.5884,E1 24.9957,E2 181.2806} C_DIS
LIN {X -5.1183,Y -110.2919,Z 117,A -96.8004,B 24.9527,C -1.5884,E1 24.9918,E2 182.6775} C_DIS
LIN {X -7.8126,Y -110.1338,Z 117,A -98.1996,B 24.9527,C -1.5884,E1 24.9879,E2 184.077} C_DIS
LIN {X -10.5026,Y -109.9098,Z 117,A -99.6055,B 24.9527,C -1.5883,E1 24.984,E2 185.484} C_DIS
LIN {X -13.2087,Y -109.6176,Z 117,A -100.9861,B 24.9527,C -1.5898,E1 24.9802,E2 186.8619} C_DIS
LIN {X -16.2096,Y -109.2156,Z 117,A -102.5542,B 24.9527,C -1.5902,E1 24.9759,E2 188.4302} C_DIS
LIN {X -18.8794,Y -108.7859,Z 117,A -103.9613,B 24.9527,C -1.5905,E1 24.972,E2 189.838} C_DIS
LIN {X -21.2317,Y -108.3499,Z 117,A -105.2328,B 24.9527,C -1.5898,E1 24.9685,E2 191.1126} C_DIS
LIN {X -24.2,Y -107.7272,Z 117,A -106.7763,B 24.9525,C -1.5917,E1 24.9643,E2 192.6534} C_DIS
LIN {X -26.6369,Y -107.1497,Z 117,A -108.0733,B 24.9525,C -1.5925,E1 24.9608,E2 193.9502} C_DIS
LIN {X -29.4491,Y -106.4122,Z 117,A -109.5921,B 24.9525,C -1.5931,E1 24.9567,E2 195.4701} C_DIS
LIN {X -31.7477,Y -105.7476,Z 117,A -110.8635,B 24.9525,C -1.5927,E1 24.9533,E2 196.7444} C_DIS
LIN {X -34.625,Y -104.8423,Z 117,A -112.4013,B 24.9523,C -1.595,E1 24.9492,E2 198.2795} C_DIS
LIN {X -37.2191,Y -103.9496,Z 117,A -113.8265,B 24.9523,C -1.5962,E1 24.9454,E2 199.7047} C_DIS
LIN {X -39.4537,Y -103.1208,Z 117,A -115.096,B 24.9523,C -1.596,E1 24.9421,E2 200.9772} C_DIS
LIN {X -41.9585,Y -102.1272,Z 117,A -116.5026,B 24.9523,C -1.5971,E1 24.9384,E2 202.3843} C_DIS
LIN {X -44.4609,Y -101.0629,Z 117,A -117.8852,B 24.952,C -1.5998,E1 24.9349,E2 203.7639} C_DIS
LIN {X -46.9223,Y -99.9439,Z 117,A -119.3199,B 24.952,C -1.6001,E1 24.9313,E2 205.2013} C_DIS
LIN {X -49.6349,Y -98.6264,Z 117,A -120.8611,B 24.9519,C -1.603,E1 24.9274,E2 206.7398} C_DIS
LIN {X -52.0485,Y -97.3744,Z 117,A -122.2766,B 24.9518,C -1.6047,E1 24.9239,E2 208.1552} C_DIS
LIN {X -54.4276,Y -96.0648,Z 117,A -123.6967,B 24.9517,C -1.6062,E1 24.9205,E2 209.5758} C_DIS
LIN {X -56.5094,Y -94.8535,Z 117,A -124.9429,B 24.9515,C -1.6082,E1 24.9175,E2 210.8211} C_DIS
LIN {X -59.0754,Y -93.2786,Z 117,A -126.5082,B 24.9515,C -1.6104,E1 24.9137,E2 212.386} C_DIS
LIN {X -61.0788,Y -91.9775,Z 117,A -127.7825,B 24.9514,C -1.611,E1 24.9108,E2 213.663} C_DIS
LIN {X -63.5652,Y -90.2788,Z 117,A -129.3213,B 24.9512,C -1.6145,E1 24.9072,E2 215.1986} C_DIS
LIN {X -65.5017,Y -88.8819,Z 117,A -130.5906,B 24.9511,C -1.6155,E1 24.9044,E2 216.47} C_DIS
LIN {X -68.3467,Y -86.7127,Z 117,A -132.4707,B 24.9509,C -1.6179,E1 24.9002,E2 218.3513} C_DIS
LIN {X -70.6907,Y -84.8128,Z 117,A -134.0724,B 24.9509,C -1.6195,E1 24.8968,E2 219.9554} C_DIS
LIN {X -73.5151,Y -82.3766,Z 117,A -135.9923,B 24.9506,C -1.6239,E1 24.8927,E2 221.8723} C_DIS
LIN {X -75.7509,Y -80.3255,Z 117,A -137.6027,B 24.9505,C -1.6257,E1 24.8894,E2 223.485} C_DIS
LIN {X -78.4421,Y -77.6995,Z 117,A -139.5288,B 24.9502,C -1.6308,E1 24.8856,E2 225.407} C_DIS
LIN {X -80.5344,Y -75.5288,Z 117,A -141.1095,B 24.95,C -1.6337,E1 24.8826,E2 226.9878} C_DIS
LIN {X -82.6124,Y -73.2517,Z 117,A -142.6778,B 24.9497,C -1.6385,E1 24.8796,E2 228.5516} C_DIS
LIN {X -84.8171,Y -70.6855,Z 117,A -144.474,B 24.9495,C -1.641,E1 24.8764,E2 230.35} C_DIS
LIN {X -86.7174,Y -68.3408,Z 117,A -146.06,B 24.9494,C -1.644,E1 24.8736,E2 231.9363} C_DIS
LIN {X -88.6763,Y -65.7823,Z 117,A -147.6888,B 24.949,C -1.6498,E1 24.8709,E2 233.5592} C_DIS
LIN {X -90.1738,Y -63.7126,Z 117,A -148.9852,B 24.9487,C -1.6542,E1 24.8688,E2 234.8512} C_DIS
LIN {X -91.6404,Y -61.5836,Z 117,A -150.4019,B 24.9487,C -1.6548,E1 24.8666,E2 236.2737} C_DIS
LIN {X -93.1191,Y -59.324,Z 117,A -151.7796,B 24.9484,C -1.6593,E1 24.8645,E2 237.6475} C_DIS
LIN {X -94.7042,Y -56.762,Z 117,A -153.3517,B 24.9482,C -1.6631,E1 24.8622,E2 239.2187} C_DIS
LIN {X -95.9093,Y -54.6982,Z 117,A -154.5996,B 24.948,C -1.6662,E1 24.8605,E2 240.4657} C_DIS
LIN {X -97.2185,Y -52.3357,Z 117,A -156.0095,B 24.9478,C -1.6697,E1 24.8586,E2 241.8746} C_DIS
LIN {X -98.4692,Y -49.9428,Z 117,A -157.4222,B 24.9475,C -1.6732,E1 24.8568,E2 243.2867} C_DIS
LIN {X -99.5036,Y -47.8475,Z 117,A -158.6869,B 24.9475,C -1.6746,E1 24.8552,E2 244.5547} C_DIS
LIN {X -100.9424,Y -44.7373,Z 117,A -160.4279,B 24.947,C -1.6811,E1 24.8532,E2 246.2899} C_DIS
LIN {X -101.8869,Y -42.5387,Z 117,A -161.7063,B 24.9469,C -1.6833,E1 24.8518,E2 247.57} C_DIS
LIN {X -102.8983,Y -40.0302,Z 117,A -163.1193,B 24.9467,C -1.6871,E1 24.8504,E2 248.982} C_DIS
LIN {X -103.8525,Y -37.4852,Z 117,A -164.4871,B 24.9463,C -1.6929,E1 24.8491,E2 250.3436} C_DIS
LIN {X -104.8735,Y -34.5286,Z 117,A -166.0918,B 24.9459,C -1.6985,E1 24.8476,E2 251.9442} C_DIS
LIN {X -105.7555,Y -31.7214,Z 117,A -167.7703,B 24.946,C -1.6974,E1 24.8462,E2 253.6351} C_DIS
LIN {X -106.6729,Y -28.4842,Z 117,A -169.4766,B 24.9456,C -1.7042,E1 24.845,E2 255.3348} C_DIS
LIN {X -107.3505,Y -25.8139,Z 117,A -170.9066,B 24.9453,C -1.7087,E1 24.844,E2 256.7626} C_DIS
LIN {X -107.9506,Y -23.1767,Z 117,A -172.2932,B 24.945,C -1.7137,E1 24.8432,E2 258.1454} C_DIS
LIN {X -108.5042,Y -20.4301,Z 117,A -173.7089,B 24.9446,C -1.7197,E1 24.8424,E2 259.5552} C_DIS
LIN {X -108.9592,Y -17.843,Z 117,A -175.1559,B 24.9446,C -1.7208,E1 24.8417,E2 261.008} C_DIS
LIN {X -109.3634,Y -15.17,Z 117,A -176.5689,B 24.9442,C -1.7249,E1 24.8412,E2 262.4198} C_DIS
LIN {X -109.7384,Y -12.177,Z 117,A -178.1164,B 24.9439,C -1.7306,E1 24.8407,E2 263.963} C_DIS
LIN {X -110.0875,Y -8.439,Z 117,A 179.892,B 24.9436,C -1.7352,E1 24.8402,E2 265.9556} C_DIS
LIN {X -110.2621,Y -5.7234,Z 117,A 178.4705,B 24.9433,C -1.7394,E1 24.84,E2 267.3756} C_DIS
LIN {X -110.3692,Y -3.0213,Z 117,A 177.0929,B 24.9429,C -1.7449,E1 24.8398,E2 268.7483} C_DIS
LIN {X -110.4102,Y -0.1303,Z 117,A 175.6064,B 24.9426,C -1.7503,E1 24.8398,E2 270.2309} C_DIS
LIN {X -110.3847,Y 2.3865,Z 117,A 174.2278,B 24.9425,C -1.7518,E1 24.8398,E2 271.6143} C_DIS
LIN {X -110.24,Y 6.1225,Z 117,A 172.2437,B 24.9422,C -1.7565,E1 24.8401,E2 273.5992} C_DIS
LIN {X -110.0052,Y 9.4686,Z 117,A 170.5525,B 24.9417,C -1.764,E1 24.8405,E2 275.2827} C_DIS
LIN {X -109.7403,Y 12.1602,Z 117,A 169.14,B 24.9414,C -1.7682,E1 24.8409,E2 276.6936} C_DIS
LIN {X -109.4496,Y 14.5349,Z 117,A 167.9379,B 24.941,C -1.7737,E1 24.8413,E2 277.8897} C_DIS
LIN {X -109.0741,Y 17.1247,Z 117,A 166.473,B 24.941,C -1.7741,E1 24.8419,E2 279.3624} C_DIS
LIN {X -108.547,Y 20.208,Z 117,A 164.8857,B 24.9406,C -1.7807,E1 24.8427,E2 280.9434} C_DIS
LIN {X -108.0194,Y 22.8607,Z 117,A 163.4733,B 24.9403,C -1.7848,E1 24.8435,E2 282.3541} C_DIS
LIN {X -107.4966,Y 25.1983,Z 117,A 162.1924,B 24.9401,C -1.7874,E1 24.8443,E2 283.6364} C_DIS
LIN {X -106.8473,Y 27.8233,Z 117,A 160.7788,B 24.9398,C -1.7915,E1 24.8452,E2 285.0486} C_DIS
LIN {X -106.0367,Y 30.7735,Z 117,A 159.2198,B 24.9394,C -1.7976,E1 24.8464,E2 286.602} C_DIS
LIN {X -105.2514,Y 33.3608,Z 117,A 157.7979,B 24.9392,C -1.8013,E1 24.8476,E2 288.0232} C_DIS
LIN {X -104.5029,Y 35.6319,Z 117,A 156.5178,B 24.939,C -1.8038,E1 24.8487,E2 289.3048} C_DIS
LIN {X -103.4924,Y 38.4724,Z 117,A 154.9732,B 24.9386,C -1.8094,E1 24.8502,E2 290.8447} C_DIS
LIN {X -102.5195,Y 40.9946,Z 117,A 153.56,B 24.9384,C -1.8133,E1 24.8516,E2 292.2565} C_DIS
LIN {X -101.4851,Y 43.4922,Z 117,A 152.1487,B 24.9381,C -1.8173,E1 24.8532,E2 293.6662} C_DIS
LIN {X -100.5181,Y 45.6791,Z 117,A 150.8986,B 24.9379,C -1.8208,E1 24.8546,E2 294.9148} C_DIS
LIN {X -99.2352,Y 48.406,Z 117,A 149.3265,B 24.9376,C -1.8251,E1 24.8565,E2 296.485} C_DIS
LIN {X -98.0007,Y 50.8592,Z 117,A 147.8909,B 24.9373,C -1.829,E1 24.8583,E2 297.9192} C_DIS
LIN {X -96.7257,Y 53.2441,Z 117,A 146.4786,B 24.937,C -1.8328,E1 24.8602,E2 299.3299} C_DIS
LIN {X -95.3926,Y 55.5973,Z 117,A 145.0651,B 24.9368,C -1.8365,E1 24.8621,E2 300.7419} C_DIS
LIN {X -94.1641,Y 57.6506,Z 117,A 143.8175,B 24.9365,C -1.8399,E1 24.8639,E2 301.9879} C_DIS
LIN {X -92.5379,Y 60.2288,Z 117,A 142.1065,B 24.9365,C -1.8394,E1 24.8665,E2 303.7086} C_DIS
LIN {X -90.656,Y 63.0225,Z 117,A 140.3963,B 24.9361,C -1.8458,E1 24.8692,E2 305.4121} C_DIS
LIN {X -88.8674,Y 65.5215,Z 117,A 138.8609,B 24.9357,C -1.8524,E1 24.8717,E2 306.9391} C_DIS
LIN {X -87.0129,Y 67.9669,Z 117,A 137.0898,B 24.9359,C -1.8499,E1 24.8748,E2 308.7247} C_DIS
LIN {X -84.9022,Y 70.583,Z 117,A 135.5055,B 24.9351,C -1.8606,E1 24.8775,E2 310.2908} C_DIS
LIN {X -83.1524,Y 72.6363,Z 117,A 134.0977,B 24.9349,C -1.8639,E1 24.8801,E2 311.6971} C_DIS
LIN {X -81.3522,Y 74.647,Z 117,A 132.6742,B 24.9347,C -1.8666,E1 24.8828,E2 313.1205} C_DIS
LIN {X -79.0961,Y 77.0356,Z 117,A 130.7806,B 24.9349,C -1.8636,E1 24.8865,E2 315.0295} C_DIS
LIN {X -76.6059,Y 79.5103,Z 117,A 129.1112,B 24.9342,C -1.8738,E1 24.8898,E2 316.6815} C_DIS
LIN {X -74.2584,Y 81.7088,Z 117,A 127.4652,B 24.9338,C -1.8786,E1 24.8931,E2 318.3228} C_DIS
LIN {X -72.2031,Y 83.5307,Z 117,A 125.8394,B 24.9342,C -1.8742,E1 24.8966,E2 319.9656} C_DIS
LIN {X -69.5027,Y 85.7889,Z 117,A 124.1652,B 24.9335,C -1.8841,E1 24.9002,E2 321.6225} C_DIS
LIN {X -66.9707,Y 87.7813,Z 117,A 122.5074,B 24.9332,C -1.8882,E1 24.9038,E2 323.2766} C_DIS
LIN {X -64.6788,Y 89.4844,Z 117,A 121.0286,B 24.9329,C -1.8914,E1 24.9071,E2 324.753} C_DIS
LIN {X -62.7274,Y 90.8612,Z 117,A 119.7841,B 24.9328,C -1.8937,E1 24.91,E2 325.9962} C_DIS
LIN {X -60.1997,Y 92.5569,Z 117,A 118.2035,B 24.9326,C -1.8967,E1 24.9137,E2 327.5749} C_DIS
LIN {X -58.1799,Y 93.8381,Z 117,A 116.9226,B 24.9325,C -1.8976,E1 24.9167,E2 328.8578} C_DIS
LIN {X -55.5962,Y 95.3932,Z 117,A 115.3801,B 24.9322,C -1.9013,E1 24.9204,E2 330.3962} C_DIS
LIN {X -53.5158,Y 96.574,Z 117,A 114.1341,B 24.9321,C -1.9033,E1 24.9234,E2 331.641} C_DIS
LIN {X -51.1351,Y 97.8554,Z 117,A 112.7259,B 24.9319,C -1.9055,E1 24.9269,E2 333.0479} C_DIS
LIN {X -48.7072,Y 99.0863,Z 117,A 111.3206,B 24.9317,C -1.9081,E1 24.9304,E2 334.4509} C_DIS
LIN {X -45.9753,Y 100.3846,Z 117,A 109.7198,B 24.9317,C -1.9092,E1 24.9344,E2 336.0528} C_DIS
LIN {X -43.5836,Y 101.4454,Z 117,A 108.3784,B 24.9315,C -1.9119,E1 24.9379,E2 337.3911} C_DIS
LIN {X -40.9845,Y 102.5235,Z 117,A 106.9131,B 24.9313,C -1.9137,E1 24.9417,E2 338.8552} C_DIS
LIN {X -38.4661,Y 103.4948,Z 117,A 105.5034,B 24.9313,C -1.9152,E1 24.9453,E2 340.2643} C_DIS
LIN {X -36.2182,Y 104.3011,Z 117,A 104.231,B 24.9313,C -1.9155,E1 24.9487,E2 341.5386} C_DIS
LIN {X -33.6579,Y 105.1552,Z 117,A 102.8552,B 24.931,C -1.9182,E1 24.9523,E2 342.9106} C_DIS
LIN {X -30.7486,Y 106.044,Z 117,A 101.2738,B 24.931,C -1.9198,E1 24.9566,E2 344.4908} C_DIS
LIN {X -28.443,Y 106.684,Z 117,A 100.0494,B 24.9308,C -1.9218,E1 24.9598,E2 345.7124} C_DIS
LIN {X -25.8077,Y 107.352,Z 117,A 98.5806,B 24.9308,C -1.9209,E1 24.9638,E2 347.1854} C_DIS
LIN {X -23.161,Y 107.954,Z 117,A 97.2029,B 24.9306,C -1.9233,E1 24.9676,E2 348.559} C_DIS
LIN {X -20.2048,Y 108.5476,Z 117,A 95.6376,B 24.9306,C -1.9246,E1 24.9719,E2 350.1231} C_DIS
LIN {X -17.8482,Y 108.9584,Z 117,A 94.3642,B 24.9306,C -1.9242,E1 24.9754,E2 351.3985} C_DIS
LIN {X -15.1748,Y 109.3627,Z 117,A 92.9559,B 24.9306,C -1.9249,E1 24.9793,E2 352.8063} C_DIS
LIN {X -12.1529,Y 109.741,Z 117,A 91.4122,B 24.9304,C -1.9273,E1 24.9835,E2 354.3454} C_DIS
LIN {X -9.4632,Y 110.0057,Z 117,A 90.0048,B 24.9304,C -1.9278,E1 24.9875,E2 355.7524} C_DIS
LIN {X -6.7675,Y 110.2044,Z 117,A 88.5976,B 24.9303,C -1.9282,E1 24.9914,E2 357.1591} C_DIS
LIN {X -4.5483,Y 110.3164,Z 117,A 87.4127,B 24.9303,C -1.9273,E1 24.9947,E2 358.3464} C_DIS
LIN {X -1.3339,Y 110.4038,Z 117,A 85.7747,B 24.9303,C -1.929,E1 24.9993,E2 359.9806} C_DIS
LIN {X 1.0557,Y 110.4055,Z 117,A 84.5325,B 24.9303,C -1.9291,E1 25.0027,E2 361.2223} C_DIS
LIN {X 4.0678,Y 110.337,Z 117,A 82.9699,B 24.9303,C -1.9293,E1 25.0071,E2 362.7842} C_DIS
LIN {X 6.7663,Y 110.2045,Z 117,A 81.5673,B 24.9303,C -1.9293,E1 25.011,E2 364.1862} C_DIS
LIN {X 9.4779,Y 110.0044,Z 117,A 80.1574,B 24.9303,C -1.9293,E1 25.0149,E2 365.5955} C_DIS
LIN {X 12.1801,Y 109.7381,Z 117,A 78.7515,B 24.9303,C -1.9292,E1 25.0188,E2 367.0007} C_DIS
LIN {X 14.555,Y 109.447,Z 117,A 77.4778,B 24.9303,C -1.9276,E1 25.0223,E2 368.2771} C_DIS
LIN {X 17.2314,Y 109.0576,Z 117,A 76.0753,B 24.9303,C -1.9272,E1 25.0262,E2 369.6791} C_DIS
LIN {X 20.1194,Y 108.5629,Z 117,A 74.5927,B 24.9303,C -1.9282,E1 25.0303,E2 371.1578} C_DIS
LIN {X 22.8733,Y 108.0167,Z 117,A 73.1309,B 24.9303,C -1.9273,E1 25.0343,E2 372.62} C_DIS
LIN {X 25.211,Y 107.4937,Z 117,A 71.8591,B 24.9305,C -1.9255,E1 25.0378,E2 373.8943} C_DIS
LIN {X 27.8363,Y 106.8439,Z 117,A 70.4571,B 24.9305,C -1.9247,E1 25.0415,E2 375.296} C_DIS
LIN {X 30.745,Y 106.045,Z 117,A 68.9228,B 24.9305,C -1.9249,E1 25.0457,E2 376.8274} C_DIS
LIN {X 34.4992,Y 104.883,Z 117,A 66.8943,B 24.9306,C -1.9238,E1 25.0511,E2 378.8549} C_DIS
LIN {X 37.2026,Y 103.9556,Z 117,A 65.4083,B 24.9307,C -1.9223,E1 25.055,E2 380.3413} C_DIS
LIN {X 39.4541,Y 103.1206,Z 117,A 64.133,B 24.9309,C -1.9199,E1 25.0583,E2 381.6196} C_DIS
LIN {X 43.5013,Y 101.4813,Z 117,A 61.9009,B 24.9309,C -1.9189,E1 25.0641,E2 383.8488} C_DIS
LIN {X 45.6887,Y 100.5138,Z 117,A 60.675,B 24.931,C -1.9182,E1 25.0672,E2 385.0735} C_DIS
LIN {X 48.4316,Y 99.2229,Z 117,A 59.0951,B 24.9312,C -1.9159,E1 25.0712,E2 386.6545} C_DIS
LIN {X 50.5483,Y 98.1597,Z 117,A 57.8201,B 24.9314,C -1.9124,E1 25.0744,E2 387.9344} C_DIS
LIN {X 53.2634,Y 96.7149,Z 117,A 56.2802,B 24.9314,C -1.9126,E1 25.0781,E2 389.4694} C_DIS
LIN {X 55.6085,Y 95.386,Z 117,A 54.8887,B 24.9315,C -1.9109,E1 25.0815,E2 390.8608} C_DIS
LIN {X 57.5556,Y 94.2219,Z 117,A 53.6609,B 24.9318,C -1.907,E1 25.0844,E2 392.094} C_DIS
LIN {X 60.1996,Y 92.557,Z 117,A 52.0947,B 24.9318,C -1.9067,E1 25.0881,E2 393.6557} C_DIS
LIN {X 62.4631,Y 91.0449,Z 117,A 50.6852,B 24.932,C -1.9045,E1 25.0914,E2 395.0657} C_DIS
LIN {X 65.3554,Y 88.989,Z 117,A 48.8178,B 24.9323,C -1.9003,E1 25.0956,E2 396.9366} C_DIS
LIN {X 67.9377,Y 87.036,Z 117,A 47.0026,B 24.9329,C -1.8914,E1 25.0997,E2 398.7662} C_DIS
LIN {X 70.5677,Y 84.915,Z 117,A 45.3983,B 24.9327,C -1.8945,E1 25.1031,E2 400.357} C_DIS
LIN {X 73.0181,Y 82.8189,Z 117,A 43.7629,B 24.9328,C -1.8928,E1 25.1066,E2 401.99} C_DIS
LIN {X 75.1586,Y 80.8825,Z 117,A 42.1007,B 24.9336,C -1.8826,E1 25.11,E2 403.6695} C_DIS
LIN {X 77.6029,Y 78.5375,Z 117,A 40.5701,B 24.9331,C -1.8888,E1 25.113,E2 405.1792} C_DIS
LIN {X 79.5032,Y 76.6132,Z 117,A 39.0945,B 24.9336,C -1.8826,E1 25.1159,E2 406.6631} C_DIS
LIN {X 81.7081,Y 74.2591,Z 117,A 37.4608,B 24.9337,C -1.8805,E1 25.119,E2 408.2945} C_DIS
LIN {X 83.6042,Y 72.1189,Z 117,A 35.8085,B 24.9345,C -1.8697,E1 25.1221,E2 409.9648} C_DIS
LIN {X 85.7715,Y 69.5241,Z 117,A 34.2061,B 24.9343,C -1.8722,E1 25.1249,E2 411.5539} C_DIS
LIN {X 87.7742,Y 66.9799,Z 117,A 32.56,B 24.9345,C -1.8696,E1 25.1277,E2 413.1985} C_DIS
LIN {X 89.2222,Y 65.0369,Z 117,A 31.2642,B 24.9348,C -1.8648,E1 25.1299,E2 414.4994} C_DIS
LIN {X 90.8554,Y 62.7357,Z 117,A 29.8543,B 24.9349,C -1.8634,E1 25.1321,E2 415.9056} C_DIS
LIN {X 92.2526,Y 60.6615,Z 117,A 28.5317,B 24.9352,C -1.859,E1 25.1342,E2 417.232} C_DIS
LIN {X 93.8198,Y 58.2092,Z 117,A 27.037,B 24.9354,C -1.8557,E1 25.1364,E2 418.7271} C_DIS
LIN {X 95.379,Y 55.6203,Z 117,A 25.5118,B 24.9356,C -1.8533,E1 25.1386,E2 420.25} C_DIS
LIN {X 96.5769,Y 53.5105,Z 117,A 24.2296,B 24.9359,C -1.8489,E1 25.1403,E2 421.536} C_DIS
LIN {X 98.2216,Y 50.4273,Z 117,A 22.3835,B 24.9364,C -1.8424,E1 25.1427,E2 423.3876} C_DIS
LIN {X 99.6825,Y 47.4752,Z 117,A 20.7259,B 24.9365,C -1.8399,E1 25.1448,E2 425.0423} C_DIS
LIN {X 100.9418,Y 44.7389,Z 117,A 19.2038,B 24.9367,C -1.8372,E1 25.1465,E2 426.5626} C_DIS
LIN {X 101.8851,Y 42.5431,Z 117,A 17.9031,B 24.9372,C -1.8309,E1 25.1479,E2 427.8709} C_DIS
LIN {X 102.9218,Y 39.9705,Z 117,A 16.5136,B 24.9373,C -1.8288,E1 25.1494,E2 429.2575} C_DIS
LIN {X 103.8472,Y 37.4998,Z 117,A 15.1825,B 24.9375,C -1.8265,E1 25.1506,E2 430.5868} C_DIS
LIN {X 104.8379,Y 34.6384,Z 117,A 13.4452,B 24.9383,C -1.8143,E1 25.1522,E2 432.3429} C_DIS
LIN {X 105.87,Y 31.3354,Z 117,A 11.7815,B 24.9383,C -1.8148,E1 25.1535,E2 433.9962} C_DIS
LIN {X 106.6847,Y 28.4406,Z 117,A 10.2558,B 24.9385,C -1.8115,E1 25.1547,E2 435.5208} C_DIS
LIN {X 107.3493,Y 25.819,Z 117,A 8.8614,B 24.9388,C -1.8075,E1 25.1556,E2 436.9164} C_DIS
LIN {X 107.9499,Y 23.1796,Z 117,A 7.4912,B 24.939,C -1.8047,E1 25.1564,E2 438.2854} C_DIS
LIN {X 108.5485,Y 20.1997,Z 117,A 5.9319,B 24.9392,C -1.8005,E1 25.1573,E2 439.8455} C_DIS
LIN {X 108.9591,Y 17.8439,Z 117,A 4.6676,B 24.9396,C -1.7955,E1 25.1579,E2 441.1141} C_DIS
LIN {X 109.3632,Y 15.1712,Z 117,A 3.2739,B 24.9398,C -1.7915,E1 25.1584,E2 442.5092} C_DIS
LIN {X 109.7381,Y 12.1799,Z 117,A 1.7488,B 24.9401,C -1.7882,E1 25.1589,E2 444.0329} C_DIS
LIN {X 109.9843,Y 9.6963,Z 117,A 0.4666,B 24.9403,C -1.7846,E1 25.1592,E2 445.316} C_DIS
LIN {X 110.205,Y 6.7559,Z 117,A -1.0514,B 24.9406,C -1.7802,E1 25.1595,E2 446.8353} C_DIS
LIN {X 110.3372,Y 4.0625,Z 117,A -2.4471,B 24.9409,C -1.7758,E1 25.1597,E2 448.2331} C_DIS
LIN {X 110.4103,Y 0.1039,Z 117,A -4.4651,B 24.9412,C -1.7708,E1 25.1597,E2 450.2509} C_DIS
LIN {X 110.3842,Y -2.4158,Z 117,A -5.8169,B 24.9416,C -1.7646,E1 25.1597,E2 451.6094} C_DIS
LIN {X 110.2921,Y -5.1138,Z 117,A -7.1968,B 24.9419,C -1.761,E1 25.1596,E2 452.9896} C_DIS
LIN {X 110.134,Y -7.8094,Z 117,A -8.5966,B 24.9422,C -1.7565,E1 25.1593,E2 454.3917} C_DIS
LIN {X 109.9101,Y -10.5003,Z 117,A -9.9927,B 24.9425,C -1.7521,E1 25.159,E2 455.7897} C_DIS
LIN {X 109.6178,Y -13.2073,Z 117,A -11.3636,B 24.9426,C -1.7494,E1 25.1585,E2 457.159} C_DIS
LIN {X 109.2152,Y -16.2124,Z 117,A -12.9211,B 24.9429,C -1.745,E1 25.1579,E2 458.7176} C_DIS
LIN {X 108.8313,Y -18.6083,Z 117,A -14.1983,B 24.9433,C -1.7401,E1 25.1573,E2 459.9988} C_DIS
LIN {X 108.3502,Y -21.2301,Z 117,A -15.5781,B 24.9435,C -1.7358,E1 25.1566,E2 461.3808} C_DIS
LIN {X 107.7319,Y -24.1791,Z 117,A -17.1016,B 24.9437,C -1.7325,E1 25.1557,E2 462.9031} C_DIS
LIN {X 107.1022,Y -26.8312,Z 117,A -18.5065,B 24.944,C -1.7284,E1 25.1548,E2 464.3096} C_DIS
LIN {X 106.4129,Y -29.4465,Z 117,A -19.9017,B 24.9443,C -1.7243,E1 25.1538,E2 465.7065} C_DIS
LIN {X 105.2357,Y -33.4091,Z 117,A -22.0253,B 24.9447,C -1.7184,E1 25.1521,E2 467.8318} C_DIS
LIN {X 104.4932,Y -35.6608,Z 117,A -23.2867,B 24.945,C -1.7132,E1 25.1509,E2 469.0984} C_DIS
LIN {X 103.4893,Y -38.4806,Z 117,A -24.7922,B 24.9452,C -1.7104,E1 25.1495,E2 470.602} C_DIS
LIN {X 102.5223,Y -40.9875,Z 117,A -26.1811,B 24.9454,C -1.7063,E1 25.1481,E2 471.9928} C_DIS
LIN {X 101.4777,Y -43.5095,Z 117,A -27.5859,B 24.9457,C -1.7025,E1 25.1466,E2 473.399} C_DIS
LIN {X 100.5098,Y -45.6976,Z 117,A -28.8232,B 24.9459,C -1.6989,E1 25.1451,E2 474.638} C_DIS
LIN {X 99.2252,Y -48.4269,Z 117,A -30.3783,B 24.9462,C -1.6946,E1 25.1433,E2 476.1949} C_DIS
LIN {X 97.9924,Y -50.875,Z 117,A -31.7893,B 24.9464,C -1.6909,E1 25.1415,E2 477.6073} C_DIS
LIN {X 96.7198,Y -53.2547,Z 117,A -33.1749,B 24.9466,C -1.6874,E1 25.1396,E2 478.9939} C_DIS
LIN {X 95.3888,Y -55.6037,Z 117,A -34.5721,B 24.9469,C -1.6834,E1 25.1377,E2 480.3931} C_DIS
LIN {X 94.1623,Y -57.6537,Z 117,A -35.8349,B 24.9472,C -1.6788,E1 25.1358,E2 481.6603} C_DIS
LIN {X 92.7903,Y -59.8361,Z 117,A -37.199,B 24.9475,C -1.6738,E1 25.1338,E2 483.0294} C_DIS
LIN {X 90.9579,Y -62.5882,Z 117,A -38.82,B 24.9475,C -1.6732,E1 25.1313,E2 484.6438} C_DIS
LIN {X 89.6234,Y -64.484,Z 117,A -40.0353,B 24.9478,C -1.6693,E1 25.1293,E2 485.8625} C_DIS
LIN {X 88.2195,Y -66.3903,Z 117,A -41.3389,B 24.9482,C -1.6626,E1 25.1271,E2 487.1755} C_DIS
LIN {X 85.9207,Y -69.34,Z 117,A -43.2517,B 24.9484,C -1.6586,E1 25.1238,E2 489.0888} C_DIS
LIN {X 84.0446,Y -71.6021,Z 117,A -44.7054,B 24.9485,C -1.6578,E1 25.1212,E2 490.5379} C_DIS
LIN {X 82.2659,Y -73.6388,Z 117,A -46.1008,B 24.9487,C -1.6545,E1 25.1186,E2 491.9348} C_DIS
LIN {X 80.3319,Y -75.744,Z 117,A -47.6531,B 24.9491,C -1.6477,E1 25.1156,E2 493.4964} C_DIS
LIN {X 77.6988,Y -78.4428,Z 117,A -49.5625,B 24.9493,C -1.6449,E1 25.1119,E2 495.4041} C_DIS
LIN {X 75.5287,Y -80.5344,Z 117,A -51.1311,B 24.9495,C -1.6409,E1 25.1087,E2 496.9756} C_DIS
LIN {X 73.1388,Y -82.7135,Z 117,A -52.9263,B 24.9501,C -1.6318,E1 25.1049,E2 498.7851} C_DIS
LIN {X 70.5599,Y -84.9214,Z 117,A -54.5345,B 24.9499,C -1.6346,E1 25.1015,E2 500.3806} C_DIS
LIN {X 67.9291,Y -87.0428,Z 117,A -56.5326,B 24.9508,C -1.62,E1 25.0971,E2 502.4056} C_DIS
LIN {X 64.3025,Y -89.7529,Z 117,A -58.6527,B 24.9505,C -1.6251,E1 25.0924,E2 504.5061} C_DIS
LIN {X 61.5643,Y -91.6535,Z 117,A -60.3462,B 24.9506,C -1.6232,E1 25.0885,E2 506.1985} C_DIS
LIN {X 59.3067,Y -93.1302,Z 117,A -61.7023,B 24.9506,C -1.6224,E1 25.0853,E2 507.5522} C_DIS
LIN {X 56.7495,Y -94.7116,Z 117,A -63.254,B 24.9508,C -1.6198,E1 25.0816,E2 509.1051} C_DIS
LIN {X 54.6882,Y -95.915,Z 117,A -64.4903,B 24.951,C -1.6176,E1 25.0786,E2 510.3427} C_DIS
LIN {X 52.328,Y -97.2227,Z 117,A -65.8851,B 24.9511,C -1.6154,E1 25.0752,E2 511.7388} C_DIS
LIN {X 49.937,Y -98.4722,Z 117,A -67.2836,B 24.9512,C -1.6131,E1 25.0717,E2 513.1388} C_DIS
LIN {X 47.4852,Y -99.6777,Z 117,A -68.8406,B 24.9517,C -1.6048,E1 25.0677,E2 514.7114} C_DIS
LIN {X 44.1662,Y -101.1914,Z 117,A -70.6855,B 24.9517,C -1.6039,E1 25.063,E2 516.5537} C_DIS
LIN {X 40.8992,Y -102.557,Z 117,A -72.3622,B 24.9515,C -1.6082,E1 25.0587,E2 518.2165} C_DIS
LIN {X 38.4222,Y -103.5108,Z 117,A -73.9464,B 24.9522,C -1.5974,E1 25.0546,E2 519.8228} C_DIS
LIN {X 35.2949,Y -104.6165,Z 117,A -75.5627,B 24.952,C -1.5997,E1 25.0503,E2 521.4304} C_DIS
LIN {X 32.3375,Y -105.5688,Z 117,A -77.1401,B 24.952,C -1.5993,E1 25.0461,E2 523.0059} C_DIS
LIN {X 29.7424,Y -106.3291,Z 117,A -78.51,B 24.952,C -1.5992,E1 25.0424,E2 524.3739} C_DIS
LIN {X 26.8272,Y -107.1033,Z 117,A -80.0717,B 24.9522,C -1.5977,E1 25.0382,E2 525.9368} C_DIS
LIN {X 23.1455,Y -107.9574,Z 117,A -82.0288,B 24.9522,C -1.596,E1 25.0329,E2 527.8952} C_DIS
LIN {X 20.1939,Y -108.5495,Z 117,A -83.5811,B 24.9523,C -1.5951,E1 25.0286,E2 529.4478} C_DIS
LIN {X 17.8398,Y -108.9598,Z 117,A -84.8106,B 24.9523,C -1.5946,E1 25.0252,E2 530.6771} C_DIS
LIN {X 15.1689,Y -109.3636,Z 117,A -86.2264,B 24.9525,C -1.593,E1 25.0213,E2 532.0954} C_DIS
LIN {X 12.1588,Y -109.7404,Z 117,A -87.7935,B 24.9525,C -1.5923,E1 25.017,E2 533.663} C_DIS
LIN {X 8.4136,Y -110.0896,Z 117,A -89.7794,B 24.9526,C -1.5899,E1 25.0114,E2 535.6535} C_DIS
LIN {X 5.7193,Y -110.2623,Z 117,A -91.1765,B 24.9526,C -1.5895,E1 25.0075,E2 537.051} C_DIS
LIN {X 1.8602,Y -110.3944,Z 117,A -93.2294,B 24.9528,C -1.5868,E1 25.0018,E2 539.1098} C_DIS
LIN {X 1.8602,Y -110.3944,Z 117,A -93.2294,B 24.9528,C -1.5868,E1 25.0018,E2 539.1098} C_DIS
Enddeposition()
LIN {X 0.8178,Y -116.4663,Z 118,A -93.0492,B 24.9567,C -1.5198,E1 25.0018,E2 539.0885} C_DIS
Startdeposition()
$VEL.CP = VEL_PRINT
LIN {X 4.4651,Y -116.3869,Z 118,A -91.0701,B 24.9562,C -1.5286,E1 25.0074,E2 537.089} C_DIS
LIN {X 7.1422,Y -116.2543,Z 118,A -89.6826,B 24.956,C -1.5322,E1 25.0113,E2 535.6934} C_DIS
LIN {X 9.9931,Y -116.044,Z 118,A -88.348,B 24.9562,C -1.5297,E1 25.015,E2 534.3655} C_DIS
LIN {X 12.838,Y -115.7638,Z 118,A -86.8732,B 24.9559,C -1.5336,E1 25.0191,E2 532.8824} C_DIS
LIN {X 15.6751,Y -115.4139,Z 118,A -85.5392,B 24.9561,C -1.5312,E1 25.0228,E2 531.5551} C_DIS
LIN {X 18.5028,Y -114.9944,Z 118,A -84.065,B 24.9558,C -1.5354,E1 25.0269,E2 530.0725} C_DIS
LIN {X 21.4943,Y -114.472,Z 118,A -82.5324,B 24.9557,C -1.5384,E1 25.0311,E2 528.5345} C_DIS
LIN {X 24.3184,Y -113.9054,Z 118,A -81.3183,B 24.9561,C -1.5304,E1 25.0344,E2 527.3409} C_DIS
LIN {X 27.0853,Y -113.2795,Z 118,A -79.9158,B 24.9561,C -1.532,E1 25.0382,E2 525.9365} C_DIS
LIN {X 29.8571,Y -112.5806,Z 118,A -78.5129,B 24.956,C -1.5333,E1 25.042,E2 524.5326} C_DIS
LIN {X 32.4402,Y -111.8647,Z 118,A -77.0481,B 24.9555,C -1.5415,E1 25.046,E2 523.0508} C_DIS
LIN {X 35.3452,Y -110.98,Z 118,A -75.6284,B 24.9555,C -1.5399,E1 25.0498,E2 521.6376} C_DIS
LIN {X 38.0582,Y -110.0792,Z 118,A -74.305,B 24.9557,C -1.5378,E1 25.0532,E2 520.3216} C_DIS
LIN {X 41.0257,Y -109.0069,Z 118,A -72.7889,B 24.9557,C -1.5383,E1 25.0572,E2 518.8077} C_DIS
LIN {X 43.4137,Y -108.0791,Z 118,A -71.4218,B 24.9553,C -1.545,E1 25.0608,E2 517.4277} C_DIS
LIN {X 46.053,Y -106.9812,Z 118,A -70.0198,B 24.9552,C -1.5469,E1 25.0644,E2 516.0246} C_DIS
LIN {X 48.6646,Y -105.8188,Z 118,A -68.6973,B 24.9552,C -1.5452,E1 25.0677,E2 514.7094} C_DIS
LIN {X 51.0872,Y -104.6717,Z 118,A -67.3042,B 24.9549,C -1.5507,E1 25.0713,E2 513.3068} C_DIS
LIN {X 53.7982,Y -103.3034,Z 118,A -65.8157,B 24.9549,C -1.553,E1 25.075,E2 511.8169} C_DIS
LIN {X 56.3172,Y -101.952,Z 118,A -64.4148,B 24.9547,C -1.5553,E1 25.0784,E2 510.4148} C_DIS
LIN {X 58.8926,Y -100.4859,Z 118,A -63.0029,B 24.9547,C -1.5558,E1 25.0818,E2 509.0059} C_DIS
LIN {X 61.2519,Y -99.0659,Z 118,A -61.6137,B 24.9544,C -1.56,E1 25.0852,E2 507.6112} C_DIS
LIN {X 63.5159,Y -97.631,Z 118,A -60.1784,B 24.9539,C -1.568,E1 25.0886,E2 506.1616} C_DIS
LIN {X 65.8928,Y -96.0428,Z 118,A -58.8302,B 24.9539,C -1.5681,E1 25.0917,E2 504.8176} C_DIS
LIN {X 68.2299,Y -94.3968,Z 118,A -57.5002,B 24.9539,C -1.5675,E1 25.0947,E2 503.4939} C_DIS
LIN {X 70.6671,Y -92.5851,Z 118,A -56.0131,B 24.9538,C -1.5704,E1 25.098,E2 502.0052} C_DIS
LIN {X 72.7796,Y -90.9352,Z 118,A -54.7007,B 24.9536,C -1.573,E1 25.1009,E2 500.6916} C_DIS
LIN {X 75.125,Y -89.0061,Z 118,A -53.2928,B 24.9536,C -1.5723,E1 25.1039,E2 499.2907} C_DIS
LIN {X 77.1539,Y -87.2545,Z 118,A -51.902,B 24.9533,C -1.5788,E1 25.1068,E2 497.8901} C_DIS
LIN {X 79.272,Y -85.3348,Z 118,A -50.503,B 24.9531,C -1.5818,E1 25.1097,E2 496.4897} C_DIS
LIN {X 81.3423,Y -83.3637,Z 118,A -49.0339,B 24.9527,C -1.5882,E1 25.1127,E2 495.0116} C_DIS
LIN {X 83.4873,Y -81.214,Z 118,A -47.6178,B 24.9527,C -1.5882,E1 25.1154,E2 493.6016} C_DIS
LIN {X 85.7421,Y -78.8281,Z 118,A -46.1661,B 24.953,C -1.5846,E1 25.1182,E2 492.1647} C_DIS
LIN {X 87.3718,Y -77.0196,Z 118,A -44.8995,B 24.9526,C -1.5909,E1 25.1205,E2 490.8888} C_DIS
LIN {X 89.2356,Y -74.8522,Z 118,A -43.4222,B 24.9522,C -1.598,E1 25.1232,E2 489.4016} C_DIS
LIN {X 90.9352,Y -72.7796,Z 118,A -42.1112,B 24.952,C -1.6012,E1 25.1255,E2 488.0892} C_DIS
LIN {X 92.8009,Y -70.3835,Z 118,A -40.6258,B 24.9517,C -1.6048,E1 25.1281,E2 486.6022} C_DIS
LIN {X 94.3968,Y -68.2299,Z 118,A -39.2452,B 24.9513,C -1.6114,E1 25.1303,E2 485.2126} C_DIS
LIN {X 96.1427,Y -65.7452,Z 118,A -37.83,B 24.9513,C -1.6119,E1 25.1326,E2 483.8034} C_DIS
LIN {X 97.8498,Y -63.1749,Z 118,A -36.5006,B 24.9516,C -1.6072,E1 25.1346,E2 482.4915} C_DIS
LIN {X 99.1603,Y -61.1008,Z 118,A -35.122,B 24.9509,C -1.6189,E1 25.1367,E2 481.0925} C_DIS
LIN {X 100.6299,Y -58.6489,Z 118,A -33.7244,B 24.9507,C -1.6226,E1 25.1387,E2 479.6933} C_DIS
LIN {X 102.0389,Y -56.1616,Z 118,A -32.327,B 24.9504,C -1.6263,E1 25.1406,E2 478.2944} C_DIS
LIN {X 103.4676,Y -53.4819,Z 118,A -30.7703,B 24.95,C -1.6338,E1 25.1426,E2 476.7283} C_DIS
LIN {X 104.7489,Y -50.9265,Z 118,A -29.5242,B 24.9502,C -1.6304,E1 25.1441,E2 475.4969} C_DIS
LIN {X 105.894,Y -48.503,Z 118,A -28.1353,B 24.9497,C -1.6377,E1 25.1458,E2 474.0981} C_DIS
LIN {X 107.0524,Y -45.8896,Z 118,A -26.7385,B 24.9495,C -1.6416,E1 25.1473,E2 472.6998} C_DIS
LIN {X 108.2138,Y -43.0768,Z 118,A -25.3329,B 24.9495,C -1.6419,E1 25.1488,E2 471.3012} C_DIS
LIN {X 109.2362,Y -40.4141,Z 118,A -23.8759,B 24.9491,C -1.6489,E1 25.1502,E2 469.8359} C_DIS
LIN {X 110.1382,Y -37.89,Z 118,A -22.5479,B 24.9488,C -1.6535,E1 25.1515,E2 468.5046} C_DIS
LIN {X 111.0349,Y -35.1757,Z 118,A -21.0812,B 24.9483,C -1.6608,E1 25.1527,E2 467.0288} C_DIS
LIN {X 112.2544,Y -31.065,Z 118,A -18.986,B 24.9479,C -1.6669,E1 25.1544,E2 464.9314} C_DIS
LIN {X 112.9829,Y -28.3007,Z 118,A -17.5895,B 24.9477,C -1.6709,E1 25.1553,E2 463.5334} C_DIS
LIN {X 113.6434,Y -25.5195,Z 118,A -16.1928,B 24.9474,C -1.675,E1 25.1562,E2 462.1352} C_DIS
LIN {X 114.2355,Y -22.7228,Z 118,A -14.8662,B 24.9474,C -1.6757,E1 25.1569,E2 460.8146} C_DIS
LIN {X 114.7881,Y -19.7368,Z 118,A -13.3826,B 24.9471,C -1.6801,E1 25.1577,E2 459.3293} C_DIS
LIN {X 115.2379,Y -16.9138,Z 118,A -12.0648,B 24.9471,C -1.6804,E1 25.1582,E2 458.0185} C_DIS
LIN {X 115.6183,Y -14.0806,Z 118,A -10.5896,B 24.9466,C -1.6883,E1 25.1587,E2 456.5335} C_DIS
LIN {X 115.929,Y -11.2389,Z 118,A -9.0919,B 24.946,C -1.6973,E1 25.1592,E2 455.0234} C_DIS
LIN {X 116.1699,Y -8.3905,Z 118,A -7.7946,B 24.946,C -1.6967,E1 25.1594,E2 453.7353} C_DIS
LIN {X 116.3332,Y -5.7151,Z 118,A -6.4174,B 24.9456,C -1.7038,E1 25.1597,E2 452.3496} C_DIS
LIN {X 116.4417,Y -2.6802,Z 118,A -5.0824,B 24.9458,C -1.701,E1 25.1597,E2 451.0289} C_DIS
LIN {X 116.4727,Y 0,Z 118,A -3.7229,B 24.9454,C -1.7073,E1 25.1597,E2 449.6628} C_DIS
LIN {X 116.4384,Y 2.8584,Z 118,A -2.2978,B 24.945,C -1.7128,E1 25.1597,E2 448.2333} C_DIS
LIN {X 116.3234,Y 5.893,Z 118,A -0.7576,B 24.9446,C -1.7199,E1 25.1595,E2 446.6856} C_DIS
LIN {X 116.1437,Y 8.746,Z 118,A 0.5037,B 24.9447,C -1.7175,E1 25.1593,E2 445.4374} C_DIS
LIN {X 115.9126,Y 11.4164,Z 118,A 1.8918,B 24.9442,C -1.725,E1 25.1589,E2 444.0397} C_DIS
LIN {X 115.5747,Y 14.4343,Z 118,A 3.2971,B 24.9442,C -1.7256,E1 25.1585,E2 442.6414} C_DIS
LIN {X 115.2128,Y 17.0902,Z 118,A 4.6853,B 24.9437,C -1.7331,E1 25.1579,E2 441.2436} C_DIS
LIN {X 114.7587,Y 19.9125,Z 118,A 6.082,B 24.9434,C -1.7371,E1 25.1573,E2 439.8456} C_DIS
LIN {X 114.2355,Y 22.7228,Z 118,A 7.4787,B 24.9432,C -1.7411,E1 25.1565,E2 438.4477} C_DIS
LIN {X 113.6434,Y 25.5195,Z 118,A 8.8757,B 24.9429,C -1.7451,E1 25.1557,E2 437.0495} C_DIS
LIN {X 112.9365,Y 28.4814,Z 118,A 10.3604,B 24.9427,C -1.7491,E1 25.1547,E2 435.5638} C_DIS
LIN {X 112.2544,Y 31.065,Z 118,A 11.6695,B 24.9424,C -1.7529,E1 25.1537,E2 434.2533} C_DIS
LIN {X 111.4054,Y 33.9807,Z 118,A 13.1537,B 24.9421,C -1.7571,E1 25.1526,E2 432.7678} C_DIS
LIN {X 110.5949,Y 36.5356,Z 118,A 14.5336,B 24.9417,C -1.764,E1 25.1514,E2 431.3794} C_DIS
LIN {X 109.6039,Y 39.4062,Z 118,A 15.948,B 24.9417,C -1.7647,E1 25.1501,E2 429.9713} C_DIS
LIN {X 108.5793,Y 42.1463,Z 118,A 17.3524,B 24.9415,C -1.7673,E1 25.1487,E2 428.5684} C_DIS
LIN {X 107.5383,Y 44.7367,Z 118,A 18.743,B 24.9411,C -1.7722,E1 25.1472,E2 427.1741} C_DIS
LIN {X 106.408,Y 47.3623,Z 118,A 20.1403,B 24.9409,C -1.7758,E1 25.1456,E2 425.7758} C_DIS
LIN {X 105.2908,Y 49.7988,Z 118,A 21.451,B 24.9407,C -1.7792,E1 25.1441,E2 424.4643} C_DIS
LIN {X 104.0369,Y 52.3678,Z 118,A 22.849,B 24.9404,C -1.7828,E1 25.1423,E2 423.0652} C_DIS
LIN {X 102.7204,Y 54.9052,Z 118,A 24.3167,B 24.94,C -1.7896,E1 25.1404,E2 421.5891} C_DIS
LIN {X 101.2533,Y 57.5641,Z 118,A 25.7318,B 24.94,C -1.79,E1 25.1385,E2 420.1806} C_DIS
LIN {X 99.9026,Y 59.8793,Z 118,A 27.0426,B 24.9397,C -1.7932,E1 25.1366,E2 418.8689} C_DIS
LIN {X 98.2487,Y 62.5535,Z 118,A 28.5399,B 24.9397,C -1.795,E1 25.1344,E2 417.375} C_DIS
LIN {X 96.7442,Y 64.8568,Z 118,A 29.8476,B 24.9395,C -1.7963,E1 25.1324,E2 416.0706} C_DIS
LIN {X 95.1234,Y 67.2115,Z 118,A 31.3253,B 24.939,C -1.8033,E1 25.13,E2 414.5837} C_DIS
LIN {X 92.6939,Y 70.526,Z 118,A 33.4064,B 24.9385,C -1.8111,E1 25.1265,E2 412.4942} C_DIS
LIN {X 90.823,Y 72.918,Z 118,A 34.8823,B 24.9383,C -1.8139,E1 25.124,E2 411.0185} C_DIS
LIN {X 89.1217,Y 74.9893,Z 118,A 36.1341,B 24.9383,C -1.8139,E1 25.1217,E2 409.7726} C_DIS
LIN {X 87.1357,Y 77.2867,Z 118,A 37.5419,B 24.9383,C -1.8133,E1 25.1192,E2 408.3725} C_DIS
Enddeposition()
END
